	6:	IF bAWrappingCone23OnAuto AND bIWrappingChannelPiston2_End AND  bIWrappingChannelPiston3_End  AND NOT bAWrap_PistRsError
		AND bAFilmLoadedCom AND NOT bAConeMissErrorAtWrpConvTemp4_24  AND NOT bAConeMissErrorAtWrpConvTemp3_24  AND NOT
		 bAConeMissErrorAtWrpConvTemp2_24 AND NOT bAConeMissErrorAtWrpConvTemp5_24 AND b2_4SetHmiSelected
		AND NOT bQSealBitAlert (*AND NOT bQSealBitAlert_24*)   AND NOT SealConeMissAlet_24 THEN
		TON_8(IN:= FALSE);
		bAWrappingCone23FwdCom:=TRUE;
		bASensorMonitorBit2:=FALSE;
 		TON_6_24(IN:=FALSE) ;
		bWrapConvStopped3_24:=FALSE;
		TON_10_24(in:=FALSE);
		step3:=step3+1;
		ELSIF  bAWrappingCone23OnAuto AND bIWrappingChannelPiston2_End AND  bIWrappingChannelPiston3_End AND NOT bAWrap_PistRsError
		AND NOT bAFilmLoadedCom AND NOT bAPauseSeq THEN
		bAFlimNotLoaded2:=TRUE;
		bAWrappingCone23OnAuto:=FALSE;
		bAWrapConeCyl23_24_1:=FALSE;
		bAPolythinSheetError:=TRUE;
		bAConeMissErrorAtWrpConvTemp4_24:=FALSE;
		bWrapConvStopped3_24:=FALSE;
 		TON_6_24(IN:=FALSE);
		TON_10_24(in:=FALSE);
		bSheetNotFeeded:='Sheet NOT Feeded'; step3:=step3+3; END_IF

	7:	step3:=step3+1;

	8:	 IF bAWrappingCone23FwdCom AND NOT bAPauseSeq  THEN
		bAWrappingCone23OnAuto:=FALSE;
		bAFilmLoadedCom:=FALSE;
		bAConeMissErrorAtWrpConvTemp4_24:=FALSE;
		 TON_6_24(IN:=FALSE) ;
		bWrapConvStopped3_24:=FALSE;
		TON_10_24(in:=FALSE);
		step3:=step3+2;
		END_IF

	9:	 IF bFilmErrClear THEN bSheetNotFeeded:='Continue Machine Operation'; bAFlimNotLoaded2:=FALSE; bASensorMonitorBit2:=FALSE;  step3:=step3+1;END_IF

	10:	 IF NOT bAPauseSeq  THEN  bAWrapConeCyl23_24_1:=FALSE;
		bA6thConeWrappOver:=TRUE;
		step3:=step3+1; END_IF

	11:	bFilmErrClear:=FALSE; TON_6_24(IN:=FALSE) ;
		bWrapConvStopped3_24:=FALSE;
		TON_10_24(in:=FALSE);step3:=step3+1;

	12:	 IF bIWrappingChannelPiston2_Home AND    bIWrappingChannelPiston3_Home   THEN
		bASet3Comp:=TRUE;
		bASet2Comp:=FALSE;
		bAWrappingCone23FwdCom:=FALSE;
		b6thConePushed_24:=TRUE;
		bAFilm1Loaded_24_6Cone:=FALSE;
		bAFilm1Loaded_24_5Cone:=FALSE;
		bASensorMonitorBit2:=FALSE;
		bAConeMissErrorAtWrpConvTemp4_24:=FALSE;
		 TON_6_24(IN:=FALSE) ;
		TON_10_24(in:=FALSE);
		bWrapConvStopped3_24:=FALSE;
		bAWrapConeCyl23_24:=FALSE;
		step3:=0;
		END_IF    sMessage_Wrapping:='Check Wrapping Piston Home  2 & 3 Reed Switch';
END_CASE


IF bAFlimNotLoaded2 AND bErrorReset AND b2_4SetHmiSelected AND bAutoModeOn THEN step3:=10; bAFlimNotLoaded2:=FALSE;HmiFilmLoadErr:=''; END_IF




                                                                             (*===============Wrapping piston 23 (Cone7,8 )on/off logic  for 2*4 model====================*)


CASE step4 OF

	0:	TON_9(IN:= FALSE);
		step4:=step4+1;

	1:	 step4:=step4+1;

	2:	IF bAutoModeOn AND  bAWrapConeCyl23_24   AND SealingOver1  AND NOT bACheckWrappConvError5 AND NOT bAFlimNotLoaded2
		AND bIWrappingChannelPiston3_Home AND bIWrappingChannelPiston2_Home AND  b2_4SetHmiSelected AND NOT bAResetEnabled
		AND NOT bAConeMissErrorAtWrpConvTemp5_24   AND b2_4SetHmiSelected  AND SealingSafety THEN
		bA8thoneReachecdWCS:=TRUE;
		TON_9(IN:= TRUE, PT:=t#1s , Q=> , ET=> );
		 sMessage_Wrapping:='Check Wrapping Piston Home 2 & 3 Reed Switch';

		IF TON_9.Q THEN  SealingOver1:=FALSE; bASensorMonitorBit3:=FALSE; step4:=step4+1; END_IF
		END_IF

	3:	 step4:=step4+1;

	4:	IF NOT bQASealingConveyorMotor AND NOT bQSealBitAlert (*AND NOT bQSealBitAlert_24 *)AND  NOT bAPauseSeq  AND  bIWrappingCone2
		AND  bIWrappingCone3   AND NOT bAConeMissErrorAtWrpConvTemp5_24  AND b2_4SetHmiSelected  AND NOT SealConeMissAlet_24
		AND SealingSafety THEN
		bAWrappingCone23OnAuto1:=TRUE;
		step4:=step4+1;
		END_IF

	5:	 step4:=step4+1;

	6:	IF bAWrappingCone23OnAuto1 AND bIWrappingChannelPiston2_End AND  bIWrappingChannelPiston3_End  AND NOT bAWrap_PistRsError
		 AND bAFilmLoadedCom AND NOT bAConeMissErrorAtWrpConvTemp5_24  AND NOT bAConeMissErrorAtWrpConvTemp3_24
		 AND NOT bAConeMissErrorAtWrpConvTemp4_24  AND NOT bAConeMissErrorAtWrpConvTemp2_24 AND NOT bQSealBitAlert (*AND NOT bQSealBitAlert_24*)
		 AND NOT SealConeMissAlet_24 THEN
		TON_9(IN:= FALSE);
		bAWrappingCone23FwdCom1:=TRUE;
		bASensorMonitorBit3:=FALSE;
		TON_8_24(IN:=FALSE);
		TON_9_24(in:=FALSE);
		bWrapConvStopped4_24:=FALSE;
		step4:=step4+1;
		ELSIF bAWrappingCone23OnAuto1 AND bIWrappingChannelPiston2_End AND  bIWrappingChannelPiston3_End  AND NOT bAWrap_PistRsError
		 AND NOT  bAFilmLoadedCom AND NOT bAPauseSeq THEN
		bAFlimNotLoaded3:=TRUE;
		bAWrappingCone23OnAuto1:=FALSE;
		bAWrapConeCyl23_24:=FALSE;
		bAPolythinSheetError:=TRUE;
		bAConeMissErrorAtWrpConvTemp5_24:=FALSE;
		bWrapConvStopped4_24:=FALSE;
 		TON_8_24(IN:=FALSE);
		TON_9_24(in:=FALSE);
		bSheetNotFeeded:='Sheet NOT Feeded'; step4:=step4+3; END_IF


	7:	step4:=step4+1;

	8:	 IF bAWrappingCone23FwdCom1 AND NOT bAPauseSeq  THEN
		bAWrappingCone23OnAuto1:=FALSE;
		bAFilmLoadedCom:=FALSE;
		bAConeMissErrorAtWrpConvTemp5_24:=FALSE;
		TON_8_24(IN:=FALSE);
		TON_9_24(in:=FALSE);
		bWrapConvStopped4_24:=FALSE;
		step4:=step4+2;
		END_IF

	9:	 IF bFilmErrClear THEN bSheetNotFeeded:='Continue Machine Operation'; bAFlimNotLoaded3:=FALSE; bASensorMonitorBit3:=FALSE;  step4:=step4+1;END_IF

	10:	 IF NOT bAPauseSeq  THEN  bAWrapConeCyl23_24:=FALSE;
		bA8thConeWrappOver:=TRUE;
		step4:=step4+1; END_IF

	11:	bFilmErrClear:=FALSE; TON_8_24(IN:=FALSE);
		TON_9_24(in:=FALSE);
		bWrapConvStopped4_24:=FALSE;step4:=step4+1;


	12:	 IF    bIWrappingChannelPiston2_Home AND    bIWrappingChannelPiston3_Home   THEN
		bASet4Comp:=TRUE;
		bASet3Comp:=FALSE;
		bAWrappingCone23FwdCom1:=FALSE;
		b8thConesPushed:=TRUE;
		bAFilm1Loaded_24_8Cone:=FALSE;
		bAFilm1Loaded_24_7Cone:=FALSE;
		bASensorMonitorBit3:=FALSE;
		bAConeMissErrorAtWrpConvTemp5_24:=FALSE;
		TON_8_24(IN:=FALSE);
		bWrapConvStopped4_24:=FALSE;
		TON_9_24(in:=FALSE);
		bAWrapConeCyl23_24:=FALSE;
		step4:=0;
		END_IF   sMessage_Wrapping:='Check Wrapping Piston Home  2 & 3 Reed Switch';
END_CASE


IF bAFlimNotLoaded3 AND b2_4SetHmiSelected AND bErrorReset AND bAutoModeOn THEN step4:=10; bAFlimNotLoaded3:=FALSE;HmiFilmLoadErr:=''; END_IF






IF bA6conesPushed AND CounterTilt23.CV<=3 THEN
bANextLayerStarted:=TRUE;
END_IF


IF bA3Pushed OR bA6conesPushed AND bAFirstConeAtWrapConv THEN
bAConvStartInterlock:=TRUE;
ELSE
bAConvStartInterlock:=FALSE;
END_IF

(*

IF bAConvFirstStartUnitB THEN
baConveyerStarted:=TRUE;
END_IF
IF baConveyerStarted AND



*)




IF bIWrappingCone1 AND   InterLockCounter.CV = 0  AND NOT  bQWrappingConveyorMotor THEN
 Interlockfor_1Cone_24:=TRUE;
 ELSE
 Interlockfor_1Cone_24:=FALSE; END_IF


IF bIWrappingCone1 AND   InterLockCounter.CV = 4  AND NOT  bQWrappingConveyorMotor THEN
 Interlockfor_5Cone_24:=TRUE;
 ELSE
 Interlockfor_5Cone_24:=FALSE; END_IF

IF bIWrappingCone1 AND   InterLockCounter.CV = 6  AND NOT  bQWrappingConveyorMotor THEN
 Interlockfor_7Cone_24:=TRUE;
 ELSE
 Interlockfor_7Cone_24:=FALSE; END_IF

WrappingCone1RT(CLK:=( bIWrappingCone1 AND NOT Interlockfor_1Cone_24 AND NOT Interlockfor_5Cone_24 AND NOT Interlockfor_7Cone_24 ), Q=> );

WrappingConvRT(CLK:= bQWrappingConveyorMotor , Q=> );

IF  WrappingConvRT.Q THEN
bAWrapConvStarted:=TRUE;

END_IF

IF WrappingCone1RT.Q THEN WCS1Sensed:=TRUE; END_IF

IF WCS1Sensed  (* AND bAWrapConvStarted OR bConvRunning*)  THEN
bAInterlockCountStart:=TRUE;
ELSE
bAInterlockCountStart:=FALSE;
 END_IF


IF  bQWrappingConveyorMotor AND NOT bIWrappingCone1 AND bAutoModeOn THEN
WCS1Sensed:=FALSE;
END_IF

(*TON_6(IN:=WCS1Sensed , PT:=T#0.2s , Q=> , ET=> );

IF TON_6.Q THEN bAWrapConvStarted:=FALSE; (*TON_6(in:=FALSE);*)END_IF


IF InterLockCounter.CV = 2 AND bManualModeOn THEN
TimerStartBit:=TRUE;
bAWrapConvStarted:=FALSE;
TON_10(IN:=TimerStartBit , PT:=t#0.2s , Q=> , ET=> );

 END_IF


IF TON_10.Q AND bQWrappingConveyorMotor THEN
bConvRunning:=TRUE;(*TON_10(in:=FALSE);*)
END_IF*)




IF bRowStopperIntOver THEN
bSaelUnitIntOverTemp:=TRUE;
END_IF



                                                                   (*=============== Interlock Logic for  2*4 WCS conveyor===================*)


CASE step7 OF


	0:	IF bSaelUnitIntOverTemp AND b2_4SetHmiSelected  THEN                                    (*========= need to check for reset Logic=    step7:=0    =======*)
		Step7:=Step7+1;
		END_IF

	1:	bWCSStart1_24:=TRUE;
		Step7:=Step7+1;

	2:	IF  bASealConvEnd1_24 THEN
		bSaelUnitIntOverTemp:=FALSE;
		Step7:=Step7+1;
		END_IF

	3:	bWCSStart2_24:=TRUE;
		bASealConvEnd1_24:=FALSE;
		Step7:=Step7+1;


	4:	IF bASealConvEnd2_24  THEN
		Step7:=Step7+1;
		END_IF

	5:	bWCSStart3_24:=TRUE;
		bASealConvEnd2_24:=FALSE;
		Step7:=2;

END_CASE



IF NOT bIEmergencySwitch OR bStopHmi  OR bServoOff OR bIMcStop THEN

bAWrappingConvStartAuto3_23:=FALSE;
bAWrappingConvStartAuto4_23:=FALSE;
bAWrappingConvStartAuto3:=FALSE;
bAWrappingConvStartAuto4:=FALSE;
bAWrappingConvStartAuto5:=FALSE;


		bAWrappingCone123FwdCom:=FALSE;


SealingOver1:=FALSE;

bAFilm1Loaded:=FALSE;
bAFilm2Loaded:=FALSE;
bAFilm3Loaded:=FALSE;
		WrapConvStartDly(in:=FALSE);
		bAConvRunning1:=FALSE;
		bWrapConvStopped2:=FALSE;
		TON_3(IN:=FALSE);
		TON_13_24(in:=FALSE);
		TON_4_24(IN:=FALSE);
		TON_12_24(in:=FALSE);
		bAConeMissErrorAtWrpConvTemp1_24:=FALSE;
		bAConeMissErrorAtWrpConvTemp2_24:=FALSE;
		bAWrapConeCyl123:=FALSE;

bWrapConvStopped2:=FALSE;
bWrapConvStopped3_24:=FALSE;
bWrapConvStopped4_24:=FALSE;
bWrapConvStopped4_24exp:=FALSE;


bAWrappingConvStart1_23:=FALSE;
bAWrappingConvStart4_23:=FALSE;
bAWrappingConvStart1:=FALSE;
bAWrappingConvStart2:=FALSE;
bAWrappingConvStart3:=FALSE;
bAWrappingConvStart4:=FALSE;
bAWrappingConvStart5:=FALSE;

bAconvReayTemp:=FALSE;
bAconvReayTemp2:=FALSE;
bAconvReadyTemp3:=FALSE;
bAconvReadyTemp4:=FALSE;
bAconvReadyTemp5:=FALSE;

bAWrappingConvStart1_23:=FALSE;
bACheckWrappConvError1:=FALSE;
bACheckWrappConvError2:=FALSE;
bACheckWrappConvError3:=FALSE;
bACheckWrappConvError4:=FALSE;
bACheckWrappConvError5:=FALSE;

bAWrappingConvStartAuto:=FALSE;
bAWrappingConvStartAuto2:=FALSE;
 bAWrappingConvStartAuto3:=FALSE;

bQAWrappingConveyorMotor1:=FALSE;
 bQAWrappingConveyorMotor2:=FALSE;
bQAWrappingConveyorMotor3:=FALSE;
 bQAWrappingConveyorMotor4:=FALSE;
bQAWrappingConveyorMotor5:=FALSE;

WrapConvStartDly3_23(IN:= FALSE);

bAConvRunning1:=FALSE;
 bAConvStartBit:=FALSE;

bASensorMonitorBit1:=FALSE;
bASensorMonitorBit2:=FALSE;
 bASensorMonitorBit3:=FALSE;

bASet1Comp:=FALSE;
bASet3Comp:=FALSE;
bASet2Comp:=FALSE;
bASet4Comp:=FALSE;

bAWrapConeCyl3:=FALSE;
bAWrapConeCyl123:=FALSE;
bAWrapConeCyl23_24_1:=FALSE;
bAWrapConeCyl23_24:=FALSE;

WCS1Sensed:=FALSE;
bSaelUnitIntOver:=FALSE;


bASealConvEnd1:=FALSE;
bASealConvEnd2:=FALSE;

InterLockCounter.RESET:=TRUE;
bAWrappingCone123OnAuto:=FALSE;
bAWrappingCone123_23OnAuto:=FALSE;
bQAWrappingConveyorMotor4_23:=FALSE;
bQAWrappingConveyorMotor3_23:=FALSE;


bCount_ConvLockBit2:=FALSE;
bCount_ConvLockBit:=FALSE;
bASealConvEnd1_24:=FALSE;
bASealConvEnd2_24:=FALSE;
step1:=0;
step2:=0;
step3:=0;
step4:=0;
step5:=0;
step6:=0;
step7:=0;
bAConvStartBit:=FALSE;

bA3Pushed:=FALSE;
b4thConePushed:=FALSE;
b6thConePushed_24:=FALSE;

bWCSStart1_24:=FALSE;
bWCSStart2_24:=FALSE;
bWCSStart3_24:=FALSE;

TON_6_24(IN:=FALSE) ;

TON_8_24(IN:=FALSE) ;
TON_9_24(IN:=FALSE);
TON_10_24(IN:=FALSE);



		bAWrappingCone3FwdCom:=FALSE;
		bAFilm1Loaded_24_4Cone:=FALSE;
		bASensorMonitorBit1:=FALSE;
		bWrapConvStopped4_24exp:=FALSE;
 		TON_5_24(IN:=FALSE);
		TON_11_24(in:=FALSE);
		bAWrappingCone3OnAuto:=FALSE;
		bAFilmLoadedCom:=FALSE;
		bAConeMissErrorAtWrpConvTemp3_24:=FALSE;
		bWrapConvStopped4_24exp:=FALSE;
		bAWrapConeCyl3:=FALSE;
		bA4thWrappOver:=FALSE;

bAWrappingCone23FwdCom:=FALSE;
		bAFilm1Loaded_24_6Cone:=FALSE;
		bAFilm1Loaded_24_5Cone:=FALSE;
		bASensorMonitorBit2:=FALSE;
		bAConeMissErrorAtWrpConvTemp4_24:=FALSE;
		 TON_6_24(IN:=FALSE) ;
		TON_10_24(in:=FALSE);
		bWrapConvStopped3_24:=FALSE;
		bAWrapConeCyl23_24:=FALSE;
		bAWrapConeCyl23_24_1:=FALSE;
		bA6thConeWrappOver:=FALSE;


		bAWrappingCone23FwdCom1:=FALSE;
		b8thConesPushed:=FALSE;
		bAFilm1Loaded_24_8Cone:=FALSE;
		bAFilm1Loaded_24_7Cone:=FALSE;
		bASensorMonitorBit3:=FALSE;
		bAConeMissErrorAtWrpConvTemp5_24:=FALSE;
		TON_8_24(IN:=FALSE);
		bWrapConvStopped4_24:=FALSE;
		TON_9_24(in:=FALSE);
		bAWrapConeCyl23_24:=FALSE;
		bAWrapConeCyl23_24:=FALSE;
		bA8thConeWrappOver:=FALSE;

ELSE
InterLockCounter.RESET:=FALSE;
END_IF
END_PROGRAM

(* POU Auto/Sealing_Conveyor_24, ST *)
PROGRAM Sealing_Conveyor_24
VAR
	bA3ConeSealStarted: BOOL;
	bA3ConeSealComp: BOOL;

	bAConeCountSenEnable1: BOOL;
	CTU_1: CTU;
	step1: INT;
	step2: INT;
	bA4thConeSealStarted: BOOL;
	bA4thConeSealComp: BOOL;

	ConvStopDly1: TON;
	bAColoumnConeDeducted: BOOL;
	step3: INT;
	bA6thConeSealStarted: BOOL;
	bA6thConeSealComp: BOOL;

	ConvStopDly2: TON;
	ConvStopDly3: TON;
	bA8thConeSealStarted: BOOL;
	bA8thConeSealComp: BOOL;
	step4: INT;

	ConvStopDly4: TON;
	bQASealingConveyor1: BOOL;
	bQASealingConveyor2: BOOL;
	bQASealingConveyor3: BOOL;
	bQASealingConveyor4: BOOL;
	Step5: INT;
	bSealConvIntOverTemp: BOOL;
	CTU_1AlarmOnly: CTU;

	bCountLockBit_24: BOOL;
	CTU_1_24: CTU;
	CTU_1_24_AlarmOnly: CTU;
	bQASealingConveyor5: BOOL;
	bQASealingConveyor6: BOOL;
	bQASealingConveyor7: BOOL;
	bQASealingConveyor8: BOOL;
	bSecSetStarted_24: BOOL;
	SealCountBit_24: BOOL;
	bCountLock1: BOOL;
	bCountLock5_24: BOOL;
	bCountLock6_24: BOOL;
	bCountLock2_24: BOOL;
	bCountLock3_24: BOOL;
	bCountLock4_24: BOOL;
	bCountLock1_24: BOOL;
	bCountLock7_24: BOOL;
	bCountLock8_24: BOOL;
	bCountLock: BOOL;
	bAConeMissAtSealConv4_24: BOOL;
	tSealStopDly_24: TIME;
	bAConeMissAtSealConv1_24: BOOL;
	bAConeMissAtSealConv2_24: BOOL;
	bAConeMissAtSealConv3_24: BOOL;
	bQASealingConveyor9: BOOL;
	bAConeMissAtSealConv5_24: BOOL;
	Timer1: TON;
	bA4ConeCrossed_24: BOOL;
	bA6ConeCrossed_24: BOOL;
	bA8ConeCrossed_24: BOOL;
	ConvStopDly01_24: TON;
	bQASealingConveyor123_24: BOOL;
	bQASealingConveyor1234_24: BOOL;
	ConvStopDly02_24: TON;
	ConvStopDly03_24: TON;
	ConvStopDly04_24: TON;
	bQASealingConveyor123456_24: BOOL;
	bQASealingConveyor12345678_24: BOOL;
	bQASealingConveyor10: BOOL;
	bQASealingConveyor11: BOOL;
	bAConeMissAtSealConv6_24: BOOL;
	bAConeMissAtSealConv7_24: BOOL;
	bQASealingConveyor12: BOOL;
	bAConeMissAtSealConv8_24: BOOL;
	bCountLock10_24: BOOL;
	bCountLock9_24: BOOL;
	bCountLock123_24: BOOL;
	bCountLock1234_24: BOOL;
	ConvStopDly06_24: TON;
	bQASealingConveyor1234_24_1: BOOL;
	bQASealingConveyor123_24_1: BOOL;
	ConvStopDly07_24: TON;
	ConvStopDly08_24: TON;
	bQASealingConveyor123456_24_1: BOOL;
	ConvStopDly09_24: TON;
	bQASealingConveyor12345678_24_1: BOOL;
	ConvStopDly11_24: TON;
	bQASealingConveyorSample123_24: BOOL;
	bQASealingConveyorSample1234_24: BOOL;
	bQASealingConveyorSample123456_24: BOOL;
	bQASealingConveyorSample12345678_24: BOOL;
	bCountLock_24: BOOL;
	bCountLock123_24_1: BOOL;
	bCountLock1234_24_1: BOOL;
	bCountLock123456_24_1: BOOL;
	bCountLock11_24: BOOL;
	bCountLock123456_24: BOOL;
	bCountLock12345678_24_1: BOOL;
	bCountLock12_24: BOOL;
	bCountLock12345678_24: BOOL;
	bSet1Started_24: BOOL;
	bSet2Started_24: BOOL;
	bSet3Started_24: BOOL;
	bSet4Started_24: BOOL;
	bCountLockBit1_24: BOOL;
	bCountLockBit2_24: BOOL;
	bCountLockBit3_24: BOOL;
	bCountLockBit4_24: BOOL;
	bAConeMissAtSealConv01_24: BOOL;
	bACounter_24Reset: BOOL;
	bACounter_24: BOOL;
END_VAR
							(*###########################Sealing Conveyor On Bit######################### *)

bQASealingConveyorMotor1:= (bQASealingConveyor1 OR bQASealingConveyor2 OR bQASealingConveyor3 OR bQASealingConveyor4 OR bQASealingConveyor5 OR bQASealingConveyor6 OR bQASealingConveyor7 OR bQASealingConveyor8 OR bQASealingConveyor9 OR bQASealingConveyor10 OR bQASealingConveyor11 OR bQASealingConveyor12 );

							(*###########################Sealing Conveyor Count interlock t######################### *)

IF bQASealingConveyorMotor AND bSet1Started_24  AND CTU_1_24_AlarmOnly.CV=3 THEN bCountLockBit1_24:=TRUE; END_IF
IF bQASealingConveyorMotor AND bSet2Started_24  AND CTU_1_24_AlarmOnly.CV=4 THEN bCountLockBit2_24:=TRUE; END_IF
IF bQASealingConveyorMotor AND bSet3Started_24  AND CTU_1_24_AlarmOnly.CV=6 THEN bCountLockBit3_24:=TRUE; END_IF
IF bQASealingConveyorMotor AND bSet4Started_24  AND CTU_1_24_AlarmOnly.CV=8 THEN bCountLockBit4_24:=TRUE; END_IF


IF bQASealingConveyorMotor AND bIConeCountSensor AND b2_4SetHmiSelected  AND NOT bCountLockBit1_24 AND NOT bCountLockBit2_24
 AND NOT bCountLockBit3_24 AND NOT bCountLockBit4_24  THEN
	bAConeCountSenEnable1:=TRUE;
ELSE
	bAConeCountSenEnable1:=FALSE;
END_IF

CTU_1(
	CU:=bAConeCountSenEnable1 ,
	RESET:= ,
	PV:=8 ,
	Q=> ,
	CV=> );


CTU_1_24_AlarmOnly(
	CU:=(bAConeCountSenEnable1 AND NOT bCountLock_24) ,
	RESET:=bACounter_24Reset OR bACounter_24 ,
	PV:=8 ,
	Q=> ,
	CV=> );


IF bQASealingConveyorMotor AND bSecSetStarted_24 AND  CTU_1.CV=8 THEN SealCountBit_24:=TRUE; END_IF


				(*############################  1,2,3rd  Cone Sealing Conveyor   ############################*)


CASE step1 OF

		0:	IF bAutoModeOn AND b2_4SetHmiSelected AND  bA3ConeWrappOver_24 AND bQASealingSeparatorYAxisPistonValve THEN
			bA3ConeSealStarted:=TRUE;
			CTU_1.RESET:=TRUE;
			bACounter_24:=TRUE;
			 tSealStopDly_24:=t#2.5s;
			ConvStopDly1(IN:=FALSE); ConvStopDly06_24(in:=FALSE);
			 step1:=step1+1; END_IF

		1:	IF NOT bAPauseSeq THEN step1:=step1+1; END_IF

		2:	IF bAutoModeOn AND b2_4SetHmiSelected AND  bA3ConeSealStarted AND bISealingSeparatorXAxisEnd THEN
			bA3ConeSealComp:=TRUE;
			CTU_1.RESET:=FALSE;
			bACounter_24:=FALSE;
		 	Timer1(IN:=FALSE);
			step1:=step1+1; END_IF

		3:	IF NOT bAPauseSeq THEN step1:=step1+1; END_IF

		4:	IF bAutoModeOn AND   bA3ConeSealComp AND (bSealConvStart1_24 OR bSealConvStart3_24)  AND NOT bASealSepaX_axisRsError THEN
			bQASealingConveyor1:=TRUE;
			ConvStopDly1(in:=FALSE);
			ConvStopDly06_24(in:=FALSE);
			bSet1Started_24:=TRUE;
			 step1:=step1+1; END_IF

		5:	ConvStopDly1(in:=FALSE);
			 step1:=step1+1;

		6:	IF NOT bAPauseSeq THEN  step1:=step1+1; END_IF

		7:	IF CTU_1_24_AlarmOnly.CV>=3 THEN
			bSealConvStart1_24:=FALSE;
			bSealConvStart3_24:=FALSE;
			bA3ConeCrossed_24:=TRUE;
			bA3ConeSealComp:=FALSE;
			bA3ConeSealStarted:=FALSE;
			 step1:=step1+1; END_IF

		8:	IF bIColumnconeDetection THEN
		step1:=step1+1;
		END_IF

		9:	ConvStopDly1(IN:=TRUE , PT:= t#0.5s , Q=> , ET=> );
			IF ConvStopDly1.Q THEN step1:=step1+1; END_IF

		10:	 step1:=step1+1;

		11:	bQASealingConveyor1:=FALSE;
			bQASealingConveyor5:=FALSE;
			bQASealingConveyor6:=FALSE;
			bA3ConeSealComp:=FALSE;
			bA3ConeSealStarted:=FALSE;
			bCountLock1_24:=FALSE;
			bCountLock5_24:=FALSE;
			bCountLock6_24:=FALSE;
			bA3ConeCrossed_24:=FALSE;
			bQASealingConveyor123_24:=FALSE;
			bAConeMissAtSealConv2_24:=FALSE;
			ConvStopDly01_24(in:=FALSE);
			bQASealingConveyorSample123_24:=FALSE;
			bQASealingConveyor123_24_1:=FALSE;
			bSet1Started_24:=FALSE;
			bCountLockBit1_24:=FALSE;
			bCountLock123_24:=FALSE;
			bCountLock123_24_1:=FALSE;
			ConvStopDly06_24(in:=FALSE);
			step1:=step1+1;


		12:	IF NOT bAPauseSeq THEN step1:=step1+1; END_IF

		13:	step1:=0;

END_CASE

				(*############################  4th Cone Sealing Conveyor   #####################*)

CASE step2 OF

	0:	IF bAutoModeOn AND b2_4SetHmiSelected AND  bA4thWrappOver AND bQASealingSeparatorYAxisPistonValve THEN
		bA4thConeSealStarted:=TRUE;
		 tSealStopDly_24:=t#2.5s;
		ConvStopDly2(IN:=FALSE);
		bQASealingConveyor123_24_1:=FALSE;
		ConvStopDly06_24(in:=FALSE);
		step2:=step2+1;
		END_IF

	1:	IF NOT bAPauseSeq THEN step2:=step2+1; END_IF

	2:	IF bAutoModeOn AND b2_4SetHmiSelected AND  bA4thConeSealStarted AND bISealingSeparatorXAxisEnd THEN
		bA4thConeSealComp:=TRUE;
		step2:=step2+1;
		END_IF

	3:	IF NOT bAPauseSeq THEN step2:=step2+1; END_IF

	4:	IF bAutoModeOn AND   bA4thConeSealComp  AND NOT bAPauseSeq THEN
		bQASealingConveyor2:=TRUE;
		bSet2Started_24:=TRUE;
		step2:=step2+1;
		END_IF

	5:	ConvStopDly2(in:=FALSE);
		ConvStopDly07_24(in:=FALSE);
		step2:=step2+1;

	6:	IF NOT bAPauseSeq THEN step2:=step2+1; END_IF

	7:	IF CTU_1_24_AlarmOnly.CV>=4 THEN
		bA4thConeSealComp:=FALSE;
		bA4thConeSealStarted:=FALSE;
		bA4ConeCrossed_24:=TRUE;
		step2:=step2+1;
		END_IF

	8:	IF NOT bAPauseSeq THEN step2:=step2+1; END_IF

	9:	IF bIColumnconeDetection THEN
		ConvStopDly2(IN:=TRUE , PT:=t#2s , Q=> , ET=> );
		IF ConvStopDly2.Q THEN    step2:=step2+1; END_IF
		END_IF

	10:	 step2:=step2+1;

	11:	bQASealingConveyor2:=FALSE;
		bQASealingConveyor9:=FALSE;
		bAColumnPushPistonStart1:=TRUE;
		bASealConvEnd1_24:=TRUE;
		bA4ConeCrossed_24:=FALSE;
		bQASealingConveyor1234_24:=FALSE;
		bAConeMissAtSealConv3_24:=FALSE;
		bAConeMissAtSealConv4_24:=FALSE;
		bQASealingConveyor10:=FALSE;
		ConvStopDly02_24(in:=FALSE);
		bQASealingConveyor9:=FALSE;
		ConvStopDly07_24(in:=FALSE);
		bQASealingConveyorSample1234_24:=FALSE;
		bQASealingConveyor1234_24_1:=FALSE;
		bSet2Started_24:=FALSE;
		bCountLockBit2_24:=FALSE;
		bCountLock1234_24_1:=FALSE;
		bCountLock1234_24:=FALSE;
		bCountLock2_24:=FALSE;
		bCountLock9_24:=FALSE;
		bCountLock10_24:=FALSE;
		step2:=0;


END_CASE


				(*############################  5,6th Cone Sealing Conveyor   #########################*)


CASE step3 OF

	0:	IF bAutoModeOn AND b2_4SetHmiSelected AND  bA6thConeWrappOver AND bQASealingSeparatorYAxisPistonValve THEN
		bA6thConeSealStarted:=TRUE;
		 tSealStopDly_24:=t#2.5s;
		ConvStopDly3(IN:=FALSE );
		bQASealingConveyor1234_24_1:=FALSE;
		ConvStopDly07_24(in:=FALSE);
		step3:=step3+1;
		END_IF

	1:	IF NOT bAPauseSeq THEN step3:=step3+1; END_IF

	2:	IF bAutoModeOn AND b2_4SetHmiSelected AND  bA6thConeSealStarted AND bISealingSeparatorXAxisEnd THEN
		bA6thConeSealComp:=TRUE;
		step3:=step3+1;
		END_IF

	3:	IF NOT bAPauseSeq THEN step3:=step3+1; END_IF

	4:	IF bAutoModeOn AND   bA6thConeSealComp AND bSealConvStart2_24 AND NOT bAPauseSeq  THEN
		bQASealingConveyor3:=TRUE;
		bSet3Started_24:=TRUE;
		step3:=step3+1;
		END_IF


	5:	ConvStopDly3(in:=FALSE);
		ConvStopDly08_24(in:=FALSE);
 		step3:=step3+1;


	6:	IF NOT bAPauseSeq THEN step3:=step3+1; END_IF

	7:	IF CTU_1_24_AlarmOnly.CV>=6 THEN
		bSealConvStart2_24:=FALSE;
		bA6ConeCrossed_24:=TRUE;
		ConvStopDly3(IN:=TRUE , PT:=t#0.5s , Q=> , ET=> );
		IF ConvStopDly3.Q THEN  step3:=step3+1; END_IF
		END_IF

	8:	 step3:=step3+1;

	9:	bA6thConeSealComp:=FALSE;
		bA6thConeSealStarted:=FALSE;
		bQASealingConveyor3:=FALSE;
		bQASealingConveyor7:=FALSE;
		bA6ConeCrossed_24:=FALSE;
		bQASealingConveyor123456_24:=FALSE;
		bAConeMissAtSealConv4_24:=FALSE;
		ConvStopDly03_24(in:=FALSE);
		bAConeMissAtSealConv6_24:=FALSE;
		bQASealingConveyor11:=FALSE;
		ConvStopDly08_24(in:=FALSE);
		bQASealingConveyorSample123456_24:=FALSE;
		bSet3Started_24:=FALSE;
		bCountLockBit3_24:=FALSE;
		bCountLock3_24:=FALSE;
		bCountLock7_24:=FALSE;
		bCountLock11_24:=FALSE;
		bCountLock123456_24:=FALSE;
		bCountLock123456_24_1:=FALSE;
		bQASealingConveyor123456_24_1:=FALSE;
		step3:=step3+1;

	10:	IF NOT bAPauseSeq THEN step3:=step3+1; END_IF

	11:	step3:=0;

END_CASE


				(*############################  7, 8th Cone Sealing Conveyor   #########################*)


CASE step4 OF

	0:	IF bAutoModeOn AND b2_4SetHmiSelected AND  bA8thConeWrappOver AND bQASealingSeparatorYAxisPistonValve THEN
		bA8thConeSealStarted:=TRUE;
		 tSealStopDly_24:=t#2.5s;
		ConvStopDly4(IN:=FALSE);
		step4:=step4+1;
		END_IF

	1:	IF NOT bAPauseSeq THEN step4:=step4+1; END_IF

	2:	IF bAutoModeOn AND b2_4SetHmiSelected AND  bA8thConeSealStarted AND bISealingSeparatorXAxisEnd THEN
		bA8thConeSealComp:=TRUE;
		step4:=step4+1;
		END_IF

	3:	IF NOT bAPauseSeq THEN step4:=step4+1; END_IF

	4:	IF bAutoModeOn AND   bA8thConeSealComp AND NOT bAPauseSeq   THEN
		bQASealingConveyor4:=TRUE;
		bSet4Started_24:=TRUE;
		step4:=step4+1;
		END_IF

	5:	ConvStopDly4(in:=FALSE);
		ConvStopDly11_24(in:=FALSE);
 		step4:=step4+1;

	6:	IF NOT bAPauseSeq THEN step4:=step4+1; END_IF

	7:	IF CTU_1_24_AlarmOnly.CV=8 THEN
		bA8thConeSealComp:=FALSE;
		bA8thConeSealStarted:=FALSE;
		bA8ConeCrossed_24:=TRUE;
		step4:=step4+1;
		END_IF

	8:	IF NOT bAPauseSeq THEN step4:=step4+1; END_IF

	9:	IF bIColumnconeDetection THEN
		ConvStopDly4(IN:=TRUE , PT:=tSealStopDly_24 , Q=> , ET=> );
		IF ConvStopDly4.Q THEN  bACounter_24:=TRUE;   step4:=step4+1; END_IF
		END_IF

	10:	 step4:=step4+1;

	11:	bQASealingConveyor4:=FALSE;
		bQASealingConveyor8:=FALSE;
		bAColumnPushPistonStart2:=TRUE;
		bASealConvEnd2_24:=TRUE;
		CTU_1.RESET:=FALSE;
		SealCountBit_24:=FALSE;
		bA8ConeCrossed_24:=FALSE;
		bQASealingConveyor12345678_24:=FALSE;
		ConvStopDly04_24(in:=FALSE);
		bAConeMissAtSealConv7_24:=FALSE;
		bQASealingConveyor12:=FALSE;
		bAConeMissAtSealConv8_24:=FALSE;
		ConvStopDly11_24(in:=FALSE);
		bQASealingConveyor12345678_24_1:=FALSE;
		bQASealingConveyorSample12345678_24:=FALSE;
		bSet4Started_24:=FALSE;
		bCountLockBit4_24:=FALSE;
		bCountLock4_24:=FALSE;
		bCountLock8_24:=FALSE;
		bCountLock12_24:=FALSE;
		bCountLock12345678_24:=FALSE;
		bCountLock12345678_24_1:=FALSE;
		step4:=0;
		bACounter_24:=FALSE;
END_CASE




IF bRowStopperIntOver  AND b2_4SetHmiSelected THEN
bSealConvIntOverTemp:=TRUE;
END_IF


CASE step5 OF


0:	IF bSealConvIntOverTemp  AND b2_4SetHmiSelected THEN
	Step5:=Step5+1;
	END_IF

1:	IF NOT bIColumnconeDetection THEN
	bSealConvStart1_24:=TRUE;
	Step5:=Step5+1;
	END_IF

2:	IF  CTU_1_24_AlarmOnly.CV=4 THEN

	Step5:=Step5+1;
	END_IF

3:	IF bIColumnconeDetection THEN
	Step5:=Step5+1;
	END_IF

4:	IF bAFirstSetToMatrix  THEN
	bSealConvStart2_24:=TRUE;
	Step5:=Step5+1;
	END_IF

5:	IF	CTU_1_24_AlarmOnly.CV=8 THEN
	bAFirstSetToMatrix:=FALSE;
	Step5:=Step5+1;
	END_IF

6:	IF bIColumnconeDetection THEN
	Step5:=Step5+1;
	END_IF

7:	IF bASecondSetToMatrix THEN
	bSealConvStart3_24:=TRUE;
	Step5:=Step5+1;
	END_IF

8:	bASecondSetToMatrix:=FALSE;
	Step5:=1;
END_CASE


(*

	IF bAresetHmi THEN
	Step5:=0;
	bSealConvStart1_24:=FALSE;
	bSealConvStart2_24:=FALSE;
	bASecondSetToMatrix:=FALSE;
	bAFirstSetToMatrix:=FALSE;
	bSealConvStart3_24:=FALSE;
	END_IF
*)

									(*--------------------------------------------------------Alarm Sequence---------------------------------------------------------*)

IF bQASealingConveyor1 AND CTU_1_24_AlarmOnly.CV =3  THEN  bCountLock1_24:=TRUE; END_IF
IF bQASealingConveyor5 AND CTU_1_24_AlarmOnly.CV =3  THEN  bCountLock5_24:=TRUE; END_IF
IF bQASealingConveyor6 AND CTU_1_24_AlarmOnly.CV =3  THEN  bCountLock6_24:=TRUE; END_IF
IF bQASealingConveyor123_24	   AND CTU_1_24_AlarmOnly.CV=3 THEN  bCountLock123_24:=TRUE; END_IF
IF bQASealingConveyor123_24_1 AND CTU_1_24_AlarmOnly.CV=3 THEN bCountLock123_24_1:=TRUE;END_IF


IF bQASealingConveyor2 AND CTU_1_24_AlarmOnly.CV =4  THEN  bCountLock2_24:=TRUE; END_IF
IF bQASealingConveyor10 AND CTU_1_24_AlarmOnly.CV =4  THEN  bCountLock10_24:=TRUE; END_IF
IF bQASealingConveyor1234_24_1 AND CTU_1_24_AlarmOnly.CV =4 THEN bCountLock1234_24_1:=TRUE; END_IF
IF bQASealingConveyor9 AND CTU_1_24_AlarmOnly.CV =4  THEN  bCountLock9_24:=TRUE; END_IF
IF bQASealingConveyor1234_24 AND CTU_1_24_AlarmOnly.CV =4  THEN  bCountLock1234_24:=TRUE; END_IF


IF bQASealingConveyor3 AND CTU_1_24_AlarmOnly.CV =6  THEN  bCountLock3_24:=TRUE; END_IF
IF bQASealingConveyor7 AND CTU_1_24_AlarmOnly.CV =6  THEN  bCountLock7_24:=TRUE; END_IF
IF bQASealingConveyor123456_24_1 AND CTU_1_24_AlarmOnly.CV =6  THEN  bCountLock123456_24_1:=TRUE; END_IF
IF bQASealingConveyor11 AND CTU_1_24_AlarmOnly.CV =6  THEN  bCountLock11_24:=TRUE; END_IF
IF bQASealingConveyor123456_24 AND CTU_1_24_AlarmOnly.CV =6  THEN  bCountLock123456_24:=TRUE; END_IF

IF bQASealingConveyor4 AND CTU_1_24_AlarmOnly.CV =8  THEN  bCountLock4_24:=TRUE; END_IF
IF bQASealingConveyor12345678_24_1 AND CTU_1_24_AlarmOnly.CV =8  THEN  bCountLock12345678_24_1:=TRUE; END_IF
IF bQASealingConveyor12 AND CTU_1_24_AlarmOnly.CV =8  THEN  bCountLock12_24:=TRUE; END_IF
IF bQASealingConveyor12345678_24 AND CTU_1_24_AlarmOnly.CV =8  THEN  bCountLock12345678_24:=TRUE; END_IF
IF bQASealingConveyor8 AND CTU_1_24_AlarmOnly.CV =8  THEN  bCountLock8_24:=TRUE; END_IF

 IF bCountLock1_24 OR bCountLock2_24 OR  bCountLock3_24 OR bCountLock4_24 OR  bCountLock5_24 OR bCountLock6_24
OR bCountLock7_24 OR bCountLock8_24 OR bCountLock9_24 OR bCountLock10_24 OR bCountLock11_24 OR bCountLock12_24
OR bCountLock123_24 OR  bCountLock1234_24  OR  bCountLock123456_24 OR  bCountLock12345678_24
OR bCountLock123_24_1 OR bCountLock1234_24_1 OR bCountLock123456_24_1 OR bCountLock12345678_24_1
THEN
 bCountLock_24:=TRUE;
 ELSE
bCountLock_24:=FALSE;
 END_IF

						(*--------------------------------------------------------Alarm Sequence Cone 2 Missing---------------------------------------------------------*)


IF bQASealingConveyor1 AND NOT bIConeCountSensor AND  NOT bAPauseSeq  THEN ConvStopDly06_24(IN:=TRUE , PT:=t#6s , Q=> , ET=> );END_IF
IF ConvStopDly06_24.Q THEN bQASealingConveyor123_24_1:=TRUE; bQASealingConveyor1:=FALSE; END_IF

IF bQASealingConveyor123_24_1    AND  (CTU_1_24_AlarmOnly.CV ) <3  AND  NOT bAPauseSeq THEN
bAConeMissAtSealConv01_24:=TRUE;
bQASealingConveyor1:=FALSE;
bQASealingConveyor123_24_1:=FALSE;
ConvStopDly06_24(in:=FALSE);
SealConeMiss:=' Cone  Missing From Sealing Conveyor';
END_IF
IF bAConeMissAtSealConv01_24 AND bErrorReset THEN
bQASealingConveyor5:=TRUE;
bAConeMissAtSealConv01_24:=FALSE;
Step1:=5;  (*tSealStopDly_24:=t#4s;*)
SealConeMiss:='Continue Machine Operation'; END_IF



						(*--------------------------------------------------------Alarm Sequence Cone 3 Missing---------------------------------------------------------*)



IF bQASealingConveyor5 OR bQASealingConveyor123_24    AND  (CTU_1_24_AlarmOnly.CV ) <3  AND  NOT bAPauseSeq  THEN
bAConeMissAtSealConv2_24:=TRUE;
bQASealingConveyor5:=FALSE;
bQASealingConveyor6:=FALSE;
bQASealingConveyor123_24:=FALSE;
ConvStopDly01_24(in:=FALSE);
bQASealingConveyorSample123_24:=FALSE;
SealConeMiss:=' Cone  Missing From Sealing Conveyor';
 END_IF
IF bAConeMissAtSealConv2_24 AND bErrorReset THEN
bQASealingConveyor6:=TRUE;  Step1:=5;  tSealStopDly_24:=t#4s;
SealConeMiss:='Continue Machine Operation'; bAConeMissAtSealConv2_24:=FALSE; END_IF

IF bQASealingConveyor6 THEN ConvStopDly01_24(IN:=TRUE , PT:=t#6s , Q=> , ET=> ); bQASealingConveyorSample123_24:=TRUE; END_IF
IF ConvStopDly01_24.Q THEN bQASealingConveyor123_24:=TRUE; END_IF



					(*--------------------------------------------------------Alarm Sequence Cone 4 Missing---------------------------------------------------------*)



IF bQASealingConveyor2 AND NOT bIConeCountSensor  AND  NOT bAPauseSeq THEN ConvStopDly07_24(IN:=TRUE , PT:=t#5s , Q=> , ET=> ); END_IF
IF ConvStopDly07_24.Q THEN bQASealingConveyor1234_24_1:=TRUE; bQASealingConveyor2:=FALSE; END_IF

IF bQASealingConveyor1234_24_1  AND  bIColumnconeDetection  AND  (CTU_1_24_AlarmOnly.CV ) <4  AND(CTU_1_24_AlarmOnly.CV ) =3 AND  NOT bAPauseSeq THEN
bAConeMissAtSealConv3_24:=TRUE;
bQASealingConveyor2:=FALSE;
bQASealingConveyor1234_24_1:=FALSE;
ConvStopDly07_24(in:=FALSE);
SealConeMiss:=' Cone  Missing From Sealing Conveyor';
END_IF
IF bAConeMissAtSealConv3_24 AND bErrorReset THEN
bQASealingConveyor10:=TRUE;
bAConeMissAtSealConv3_24:=FALSE;
Step2:=5;  tSealStopDly_24:=t#4s;
SealConeMiss:='Continue Machine Operation'; END_IF


IF bQASealingConveyor10 OR bQASealingConveyor1234_24 AND  bIColumnconeDetection  AND  (CTU_1_24_AlarmOnly.CV ) <4 AND (CTU_1_24_AlarmOnly.CV ) =3 AND  NOT bAPauseSeq   THEN
bAConeMissAtSealConv4_24:=TRUE;
bQASealingConveyor10:=FALSE;
bQASealingConveyor1234_24:=FALSE;
ConvStopDly02_24(in:=FALSE);
bQASealingConveyor9:=FALSE;
bQASealingConveyorSample1234_24:=FALSE;
SealConeMiss:=' Cone  Missing From Sealing Conveyor';
 END_IF
IF bAConeMissAtSealConv4_24 AND bErrorReset THEN
bQASealingConveyor9:=TRUE;  Step2:=5;  tSealStopDly_24:=t#4s;
SealConeMiss:='Continue Machine Operation'; bAConeMissAtSealConv4_24:=FALSE; END_IF

IF bQASealingConveyor9 THEN ConvStopDly02_24(IN:=TRUE , PT:=t#6s , Q=> , ET=> ); bQASealingConveyorSample1234_24:=TRUE;END_IF
IF ConvStopDly02_24.Q THEN bQASealingConveyor1234_24:=TRUE; END_IF



					(*--------------------------------------------------------Alarm Sequence Cone 6 Missing---------------------------------------------------------*)


IF bQASealingConveyor3 AND NOT bIConeCountSensor  AND  NOT bAPauseSeq THEN ConvStopDly08_24(IN:=TRUE , PT:=t#5s , Q=> , ET=> ); END_IF
IF ConvStopDly08_24.Q THEN bQASealingConveyor123456_24_1:=TRUE; bQASealingConveyor3:=FALSE; END_IF

IF bQASealingConveyor123456_24_1    AND  (CTU_1_24_AlarmOnly.CV ) <6  AND  (CTU_1_24_AlarmOnly.CV ) >=4  AND  NOT bAPauseSeq THEN
bAConeMissAtSealConv5_24:=TRUE;
bQASealingConveyor3:=FALSE;
ConvStopDly08_24(in:=FALSE);
bQASealingConveyor123456_24_1:=FALSE;
SealConeMiss:=' Cone  Missing From Sealing Conveyor';
END_IF
IF bAConeMissAtSealConv5_24 AND bErrorReset THEN
bQASealingConveyor11:=TRUE;
bAConeMissAtSealConv5_24:=FALSE;
Step3:=5;  tSealStopDly_24:=t#4s;
SealConeMiss:='Continue Machine Operation';
END_IF

IF bQASealingConveyor11  OR bQASealingConveyor123456_24   AND  (CTU_1_24_AlarmOnly.CV ) <6 AND  (CTU_1_24_AlarmOnly.CV ) >=4 AND  NOT bAPauseSeq   THEN
bAConeMissAtSealConv6_24:=TRUE;
bQASealingConveyor11:=FALSE;
bQASealingConveyor123456_24:=FALSE;
ConvStopDly03_24(in:=FALSE);
bQASealingConveyor7:=FALSE;
bQASealingConveyorSample123456_24:=FALSE;
SealConeMiss:=' Cone  Missing From Sealing Conveyor';
 END_IF
IF bAConeMissAtSealConv6_24 AND bErrorReset THEN
bQASealingConveyor7:=TRUE;  Step3:=5;  tSealStopDly_24:=t#4s;
SealConeMiss:='Continue Machine Operation'; bAConeMissAtSealConv6_24:=FALSE; END_IF

IF bQASealingConveyor7 THEN ConvStopDly03_24(IN:=TRUE , PT:=t#6s , Q=> , ET=> ); bQASealingConveyorSample123456_24:=TRUE;END_IF
IF ConvStopDly03_24.Q THEN bQASealingConveyor123456_24:=TRUE; END_IF


		                            (*--------------------------------------------------------Alarm Sequence Cone 8 Missing---------------------------------------------------------*)


IF bQASealingConveyor4 AND NOT bIConeCountSensor  AND  NOT bAPauseSeq THEN ConvStopDly11_24(IN:=TRUE , PT:=t#5s , Q=> , ET=> ); END_IF
IF ConvStopDly11_24.Q THEN bQASealingConveyor12345678_24_1:=TRUE; bQASealingConveyor4:=FALSE; END_IF


IF bQASealingConveyor12345678_24_1  AND  bIColumnconeDetection  AND  (CTU_1_24_AlarmOnly.CV ) <8 AND  (CTU_1_24_AlarmOnly.CV ) >=6  AND  NOT bAPauseSeq THEN
bAConeMissAtSealConv7_24:=TRUE;
bQASealingConveyor4:=FALSE;
ConvStopDly11_24(in:=FALSE);
bQASealingConveyor12345678_24_1:=FALSE;
SealConeMiss:=' Cone  Missing From Sealing Conveyor';
END_IF
IF bAConeMissAtSealConv7_24 AND bErrorReset THEN
bQASealingConveyor12:=TRUE;
bAConeMissAtSealConv7_24:=FALSE;
Step4:=5;  tSealStopDly_24:=t#4s;
SealConeMiss:='Continue Machine Operation'; END_IF


IF bQASealingConveyor12 OR bQASealingConveyor12345678_24  AND  bIColumnconeDetection  AND  (CTU_1_24_AlarmOnly.CV ) <8 AND  (CTU_1_24_AlarmOnly.CV ) >=6
AND  NOT bAPauseSeq THEN
bAConeMissAtSealConv8_24:=TRUE;
bQASealingConveyor12:=FALSE;
bQASealingConveyor12345678_24:=FALSE;
ConvStopDly04_24(in:=FALSE);
bQASealingConveyor8:=FALSE;
bQASealingConveyorSample12345678_24:=FALSE;
SealConeMiss:=' Cone  Missing From Sealing Conveyor';
 END_IF
IF bAConeMissAtSealConv8_24 AND bErrorReset THEN
bQASealingConveyor8:=TRUE;  Step4:=5;  tSealStopDly_24:=t#4s;
SealConeMiss:='Continue Machine Operation'; bAConeMissAtSealConv8_24:=FALSE; END_IF

IF bQASealingConveyor8 THEN ConvStopDly04_24(IN:=TRUE , PT:=t#6s , Q=> , ET=> ); bQASealingConveyorSample12345678_24:=TRUE; END_IF
IF ConvStopDly04_24.Q THEN bQASealingConveyor12345678_24:=TRUE; END_IF



									(*##############################Alarm Sequence in HMI#################################*)


IF bAConeMissAtSealConv01_24 OR bAConeMissAtSealConv2_24 OR bAConeMissAtSealConv3_24 OR bAConeMissAtSealConv8_24
OR bAConeMissAtSealConv4_24 OR bAConeMissAtSealConv5_24 OR bAConeMissAtSealConv6_24 OR bAConeMissAtSealConv7_24  THEN
 bQSealBitAlert:=TRUE; END_IF

IF bQSealBitAlert   AND bErrorReset   THEN   bQSealBitAlert:=FALSE; END_IF

IF bQASealingConveyor123_24_1 OR  bQASealingConveyor123_24 OR bQASealingConveyor1234_24_1 OR bQASealingConveyor123456_24_1
OR bQASealingConveyor12345678_24 OR bQASealingConveyorSample12345678_24 OR bQASealingConveyorSample123456_24 OR
 bQASealingConveyorSample1234_24 OR bQASealingConveyorSample123_24 THEN
  bQSealBitAlert_24:=TRUE; ELSE  bQSealBitAlert_24:=FALSE;  END_IF

IF bQASealingConveyor1 OR bQASealingConveyor2 OR bQASealingConveyor3 OR bQASealingConveyor4 OR bQASealingConveyor5 OR
bQASealingConveyor6 OR bQASealingConveyor7 OR bQASealingConveyor8 OR bQASealingConveyor9 OR bQASealingConveyor10 OR
bQASealingConveyor11 OR bQASealingConveyor12   THEN SealConeMissAlet_24:= TRUE; ELSE SealConeMissAlet_24:= FALSE; END_IF



IF NOT bIEmergencySwitch OR bStopHmi  OR bServoOff OR bIMcStop THEN
bQSealBitAlert:=FALSE;
bQSealBitAlert_24:=FALSE;
bACounter_24Reset:=TRUE;
CTU_1.RESET:=TRUE;

bAConeMissAtSealConv01_24:=FALSE;
bAConeMissAtSealConv2_24 :=FALSE;
bAConeMissAtSealConv3_24:=FALSE;
bAConeMissAtSealConv4_24:=FALSE;
bAConeMissAtSealConv5_24:=FALSE;
bAConeMissAtSealConv6_24:=FALSE;
bAConeMissAtSealConv7_24:=FALSE;
bAConeMissAtSealConv8_24:=FALSE;

bQASealingConveyor1:=FALSE;
bQASealingConveyor2:=FALSE;
bQASealingConveyor3:=FALSE;
bQASealingConveyor4:=FALSE;
bQASealingConveyor5:=FALSE;
bQASealingConveyor6:=FALSE;
bQASealingConveyor7:=FALSE;
bQASealingConveyor8:=FALSE;
bQASealingConveyor9:=FALSE;
bQASealingConveyor10:=FALSE;
bQASealingConveyor11:=FALSE;
bQASealingConveyor12:=FALSE;

bQASealingConveyor123_24:=FALSE;
bQASealingConveyor1234_24:=FALSE;
bQASealingConveyor123456_24:=FALSE;
bQASealingConveyor12345678_24:=FALSE;

bQASealingConveyor123_24_1:=FALSE;
 bQASealingConveyor1234_24_1:=FALSE;
 bQASealingConveyor123456_24_1:=FALSE;
 bQASealingConveyor12345678_24_1:=FALSE;

bQASealingConveyorSample123_24 :=FALSE;
bQASealingConveyorSample1234_24 :=FALSE;
bQASealingConveyorSample123456_24 :=FALSE;
bQASealingConveyorSample12345678_24:=FALSE;

bCountLock1_24:=FALSE;
bCountLock2_24:=FALSE;
bCountLock3_24:=FALSE;
bCountLock4_24:=FALSE;
bCountLock5_24:=FALSE;
bCountLock6_24:=FALSE;
bCountLock7_24:=FALSE;
bCountLock8_24:=FALSE;
bCountLock9_24:=FALSE;
bCountLock10_24:=FALSE;
bCountLock11_24:=FALSE;
bCountLock12_24:=FALSE;

bCountLock123_24:=FALSE;
bCountLock1234_24:=FALSE;
bCountLock123456_24:=FALSE;
bCountLock12345678_24:=FALSE;

bCountLock123_24_1:=FALSE;
bCountLock1234_24_1:=FALSE;
bCountLock123456_24_1:=FALSE;
bCountLock12345678_24_1:=FALSE;

bCountLockBit1_24:=FALSE;
bCountLockBit2_24:=FALSE;
bCountLockBit3_24:=FALSE;
bCountLockBit4_24:=FALSE;

Step1:=0;
Step2:=0;
Step3:=0;
Step4:=0;
Step5:=0;

bCountLock_24:=FALSE;

ConvStopDly1(IN:=FALSE);
ConvStopDly2(IN:=FALSE);
ConvStopDly3(IN:=FALSE);
ConvStopDly4(IN:=FALSE);

ConvStopDly01_24(in:=FALSE);
ConvStopDly02_24(in:=FALSE);
ConvStopDly03_24(in:=FALSE);
ConvStopDly04_24(in:=FALSE);
ConvStopDly06_24(in:=FALSE);
ConvStopDly07_24(in:=FALSE);
ConvStopDly08_24(in:=FALSE);
ConvStopDly09_24(in:=FALSE);
ConvStopDly11_24(in:=FALSE);

bSet1Started_24:=FALSE;
bSet2Started_24:=FALSE;
bSet3Started_24:=FALSE;
bSet4Started_24:=FALSE;

bSealConvStart1_24:=FALSE;
bSealConvStart2_24:=FALSE;
bSealConvStart3_24:=FALSE;


bA3ConeCrossed_24:=FALSE;
bA4ConeCrossed_24:=FALSE;
bA6ConeCrossed_24:=FALSE;
bA8ConeCrossed_24:=FALSE;


bA3ConeSealComp:=FALSE;
bA4thConeSealComp:=FALSE;
bA6thConeSealComp:=FALSE;
bA8thConeSealComp:=FALSE;

bA3ConeSealStarted:=FALSE;
bA4thConeSealStarted:=FALSE;
bA6thConeSealStarted:=FALSE;
bA8thConeSealStarted:=FALSE;




ELSE
bACounter_24Reset:=FALSE;
CTU_1.RESET:=FALSE;
END_IF
END_PROGRAM

(* POU ERROR_1, ST *)
PROGRAM ERROR_1
VAR
	bfAlarmbit1: BOOL;
	sAlarmBuffer: ARRAY[1..5] OF STRING;
	sAlarmArray: ARRAY[0..50] OF STRING;
	ifAlarmStep: INT;
	k: INT;
	sAlarmValue: STRING;
	bfAlarmGenerated: BOOL;
	sAlarm1: STRING(80);
	bfAlarmbit2: BOOL;
	bfAlarmbit3: BOOL;
	bfAlarmbit4: BOOL;
	bfAlarmbit5: BOOL;
	sAlarm2: STRING(80);
	sAlarm3: STRING(80);
	sAlarm4: STRING(80);
	sAlarm5: STRING(80) ;
	ifAlarmMoveStep: INT;
	bfReset: BOOL;
	ifAlarmStepClear: INT;
	bClearAlarm: BOOL;
	bDoIndex: BOOL;
	R_TRIG1: R_TRIG;
	Berror: BOOL;




	bRetIUniitAHomeNok: BOOL;
	bRetreivalUnitHomNok: BOOL;
	bRetIUniitBHomeNok: BOOL;
END_VAR
(*============Reteival Unit Error Messages================== *)


	IF bAutoModeOn AND bMCStartInAuto AND bIUnitA_StartPB AND NOT bIUnitA_RowStopperHome AND NOT bUnitARowStopperStarted  THEN bRetIUniitAHomeNok:=TRUE; ELSE  bRetIUniitAHomeNok:=FALSE; END_IF

	IF bAutoModeOn AND bMCStartInAuto AND bIUnitB_StartPB AND NOT bIUnitB_RowStopperHome AND NOT bUnitBRowStopperStarted THEN bRetIUniitBHomeNok:=TRUE; ELSE  bRetIUniitBHomeNok:=FALSE; END_IF

	IF bRetIUniitAHomeNok OR bRetIUniitAHomeNok THEN bRetreivalUnitHomNok:=TRUE; ELSE bRetreivalUnitHomNok:=FALSE; END_IF


















(*

IF bfAlarmbit1 THEN sAlarmBuffer[1]:=sAlarm1;bfAlarmbit1:=FALSE; END_IF
IF bfAlarmbit2 THEN sAlarmBuffer[2]:=sAlarm2;bfAlarmbit2:=FALSE; END_IF
IF bfAlarmbit3 THEN sAlarmBuffer[3]:=sAlarm3;bfAlarmbit3:=FALSE; END_IF
IF bfAlarmbit4 THEN sAlarmBuffer[4]:=sAlarm4;bfAlarmbit4:=FALSE; END_IF
IF bfAlarmbit5 THEN sAlarmBuffer[5]:=sAlarm5;bfAlarmbit5:=FALSE; END_IF
*)
CASE ifAlarmMoveStep OF

	0:	IF sAlarmBuffer[1]<>'' THEN ifAlarmMoveStep:=1;
			ELSIF sAlarmBuffer[2]<>'' THEN ifAlarmMoveStep:=3;
			ELSIF sAlarmBuffer[3]<>'' THEN ifAlarmMoveStep:=5;
			ELSIF sAlarmBuffer[4]<>'' THEN ifAlarmMoveStep:=7;
			ELSIF sAlarmBuffer[5]<>'' THEN ifAlarmMoveStep:=9;
		END_IF

	1:	sAlarmValue:=sAlarmBuffer[1];bfAlarmGenerated:=TRUE;ifAlarmMoveStep:=ifAlarmMoveStep+1;

	2:	IF NOT bfAlarmGenerated AND NOT bfAlarmbit1 THEN sAlarm1:=sAlarmBuffer[1]:='';ifAlarmMoveStep:=0; END_IF

	3:	sAlarmValue:=sAlarmBuffer[2];bfAlarmGenerated:=TRUE;ifAlarmMoveStep:=ifAlarmMoveStep+1;

	4:	IF NOT bfAlarmGenerated THEN sAlarm2:=sAlarmBuffer[2]:='';ifAlarmMoveStep:=0; END_IF

	5:	sAlarmValue:=sAlarmBuffer[3];bfAlarmGenerated:=TRUE;ifAlarmMoveStep:=ifAlarmMoveStep+1;

	6:	IF NOT bfAlarmGenerated THEN sAlarm3:=sAlarmBuffer[3]:='';ifAlarmMoveStep:=0; END_IF

	7:	sAlarmValue:=sAlarmBuffer[4];bfAlarmGenerated:=TRUE;ifAlarmMoveStep:=ifAlarmMoveStep+1;

	8:	IF NOT bfAlarmGenerated THEN sAlarm4:=sAlarmBuffer[4]:='';ifAlarmMoveStep:=0; END_IF

	9:	sAlarmValue:=sAlarmBuffer[5];bfAlarmGenerated:=TRUE;ifAlarmMoveStep:=ifAlarmMoveStep+1;

	10:	IF NOT bfAlarmGenerated THEN sAlarm5:=sAlarmBuffer[5]:='';ifAlarmMoveStep:=0; END_IF

END_CASE






IF bfAlarmGenerated THEN
CASE ifAlarmStep OF

	0: 	k:=50;ifAlarmStep:=ifAlarmStep+1;

	1:	sAlarmArray[k]:=sAlarmArray[k-1];ifAlarmStep:=ifAlarmStep+1;

	2: 	IF NOT (k=1) THEN k:=k-1;ifAlarmStep:=1; ELSE ifAlarmStep:=ifAlarmStep+1; END_IF

	3:	sAlarmArray[0]:=sAlarmValue;ifAlarmStep:=ifAlarmStep+1;

	4:	bfAlarmGenerated:=FALSE;ifAlarmStep:=0;

END_CASE
END_IF
(*
 IF bClearAlarm THEN
FOR i:=0 TO 50 DO
	sAlarmArray[i]:='';
END_FOR
END_IF
*)
IF bFeedinfCylFwdRsError THEN sAlarmBuffer[1]:='chect Cone Feeding Piston Fwd Reed Switdh'; ELSE sAlarmBuffer[1]:=''; END_IF
IF bfAlarmbit2 THEN sAlarmBuffer[2]:=sAlarm2;ELSE sAlarmBuffer[2]:=''; END_IF
IF bfAlarmbit3 THEN sAlarmBuffer[3]:=sAlarm3;ELSE sAlarmBuffer[3]:=''; END_IF
IF bfAlarmbit4 THEN sAlarmBuffer[4]:=sAlarm4;ELSE sAlarmBuffer[4]:=''; END_IF
IF bfAlarmbit5 THEN sAlarmBuffer[5]:=sAlarm5;ELSE sAlarmBuffer[5]:=''; END_IF

IF bfAlarmbit1 OR bfAlarmbit2 OR bfAlarmbit3 OR bfAlarmbit4 OR bfAlarmbit5 THEN
Berror:=TRUE;
ELSE
Berror:=FALSE;
END_IF
END_PROGRAM

(* Visualisation AA
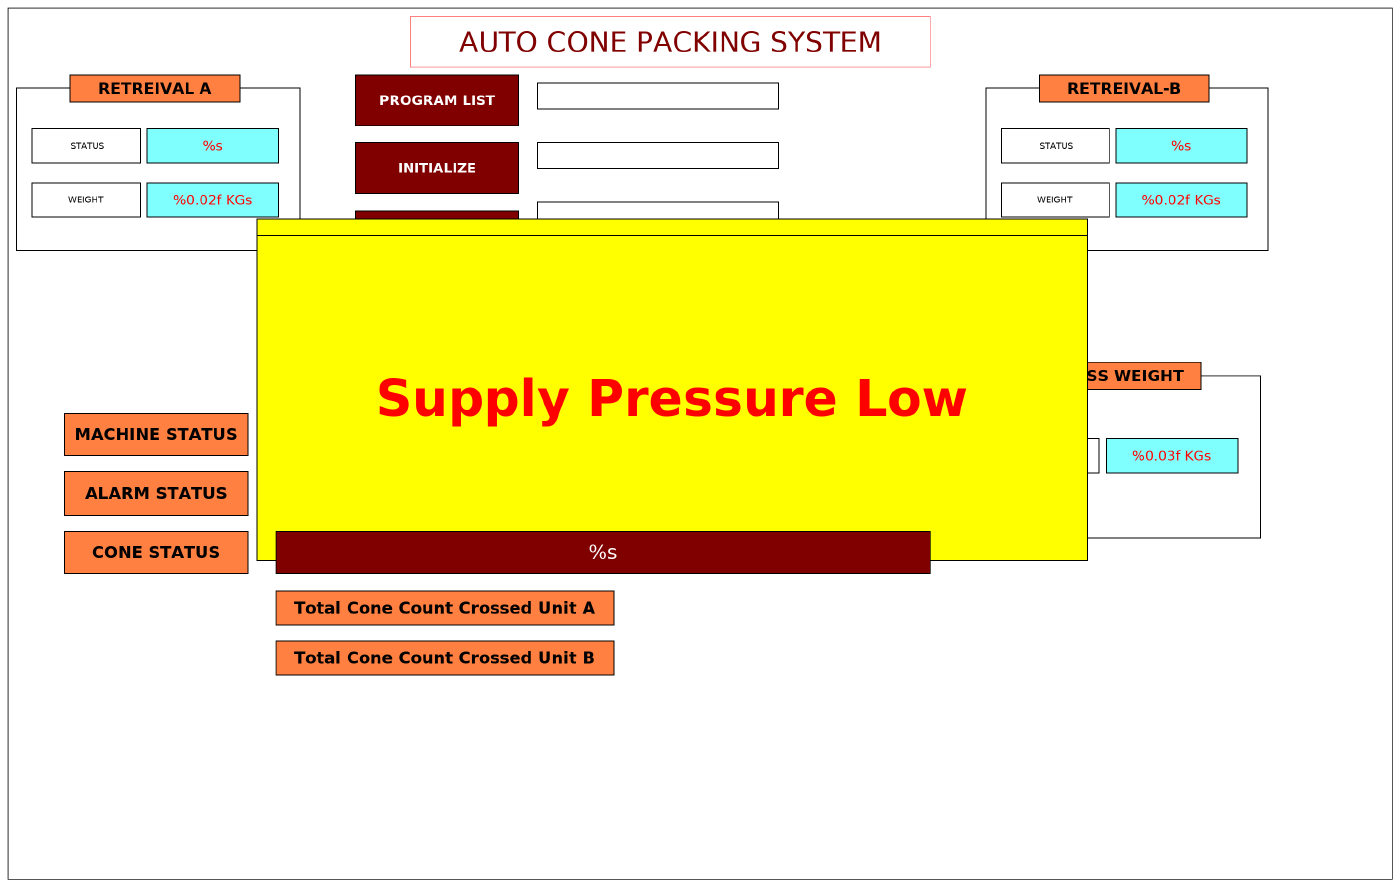
group at (10,0)-(1441,901)
  rounded rectangle at (289,56)-(425,99): text "PROGRAM LIST"; opens Models
  rounded rectangle at (289,113)-(425,156): text "INITIALIZE"; alarm colour if bAInitializeSeq; taps bInitializeHmi
  rounded rectangle at (289,290)-(425,333): text "STOP"; alarm colour if bStopHmi; taps bStopHmi
  rounded rectangle at (440,63)-(641,85): text "PROGRAM NO"
  rounded rectangle at (440,113)-(641,135): text "DETAILS"
  rounded rectangle at (440,163)-(641,185): text "NO OF CONE PROCESSED"
  rounded rectangle at (440,219)-(641,241): text "NO OF CARTONS PROCESSED"
  rounded rectangle at (440,269)-(641,291): text "DATE"
  rounded rectangle at (335,7)-(767,50): text "AUTO CONE PACKING SYSTEM"
  rounded rectangle at (289,170)-(425,213): text "PAUSE"; alarm colour if bAPauseSeq; taps bPauseHmi
  rounded rectangle at (289,226)-(425,270): text "RESUME"; alarm colour if bAPauseSeq; taps bResumeHmi
  rounded rectangle at (47,340)-(200,376): text "MACHINE STATUS"
  rounded rectangle at (47,389)-(200,426): text "ALARM STATUS"
  rounded rectangle at (223,389)-(767,426): text "%s"; shows sMianAlarmStatus
  group at (7,56)-(243,204)
    rounded rectangle at (56,0)-(233,33): text "RETREIVAL A"
    rounded rectangle at (136,64)-(273,105): text "%s"; shows sRetreivalAStatus
    rounded rectangle at (16,64)-(129,105): text "STATUS"
    rounded rectangle at (16,128)-(129,169): text "WEIGHT"
    rounded rectangle at (136,128)-(273,169): text "%0.02f KGs"; shows rRetUnitAWeight
  group at (813,56)-(1048,204)
    rounded rectangle at (56,0)-(233,33): text "RETREIVAL-B"
    rounded rectangle at (136,64)-(273,105): text "%s"; shows sRetreivalBStatus
    rounded rectangle at (16,64)-(129,105): text "STATUS"
    rounded rectangle at (16,128)-(129,169): text "WEIGHT"
    rounded rectangle at (136,128)-(273,169): text "%0.02f KGs"; shows rRetUnitBWeight
  group at (279,248)-(751,397)
    rounded rectangle at (0,0)-(591,211): invisible if not bHidePopUp
    rounded rectangle at (140,110)-(251,161): text "YES"; invisible if NOT bHidePopUp; taps bPauseYesHmi
    rounded rectangle at (320,110)-(431,161): text "NO"; invisible if not bHidePopUp; taps bPauseNoHmi
    rounded rectangle at (88,16)-(513,73): text "Machine is Running. Do You Want to Change / Mode to Manual ?"; invisible if NOT bHidePopUp
    rounded rectangle at (48,168)-(553,201): text "NOTE:- All the Operations will be Aborted."; invisible if NOT bHidePopUp
  rounded rectangle at (223,340)-(767,376): text "%s"; shows sMCStatus
  group at (806,297)-(1042,445)
    rounded rectangle at (56,0)-(233,33): text "GROSS WEIGHT"
    rounded rectangle at (14,91)-(127,132): text "WEIGHT"
    rounded rectangle at (134,91)-(271,132): text "%0.03f KGs"; shows rGrossWeight
  rounded rectangle at (207,177)-(898,450): text "Emergency Pressed"; invisible if NOT bAEmergencyPressed
  rounded rectangle at (207,191)-(898,464): text "Supply Pressure Low"; invisible if NOT bASupplyPressureError
  rounded rectangle at (223,489)-(504,518): text "Total Cone Count Crossed Unit A"
  rounded rectangle at (223,531)-(504,560): text "Total Cone Count Crossed Unit B"
  rounded rectangle at (47,439)-(200,475): text "CONE STATUS"
  rounded rectangle at (223,439)-(767,475): text "%s"; shows Message1_24
4 more shapes without text or variables
*)

(* Visualisation ALARM
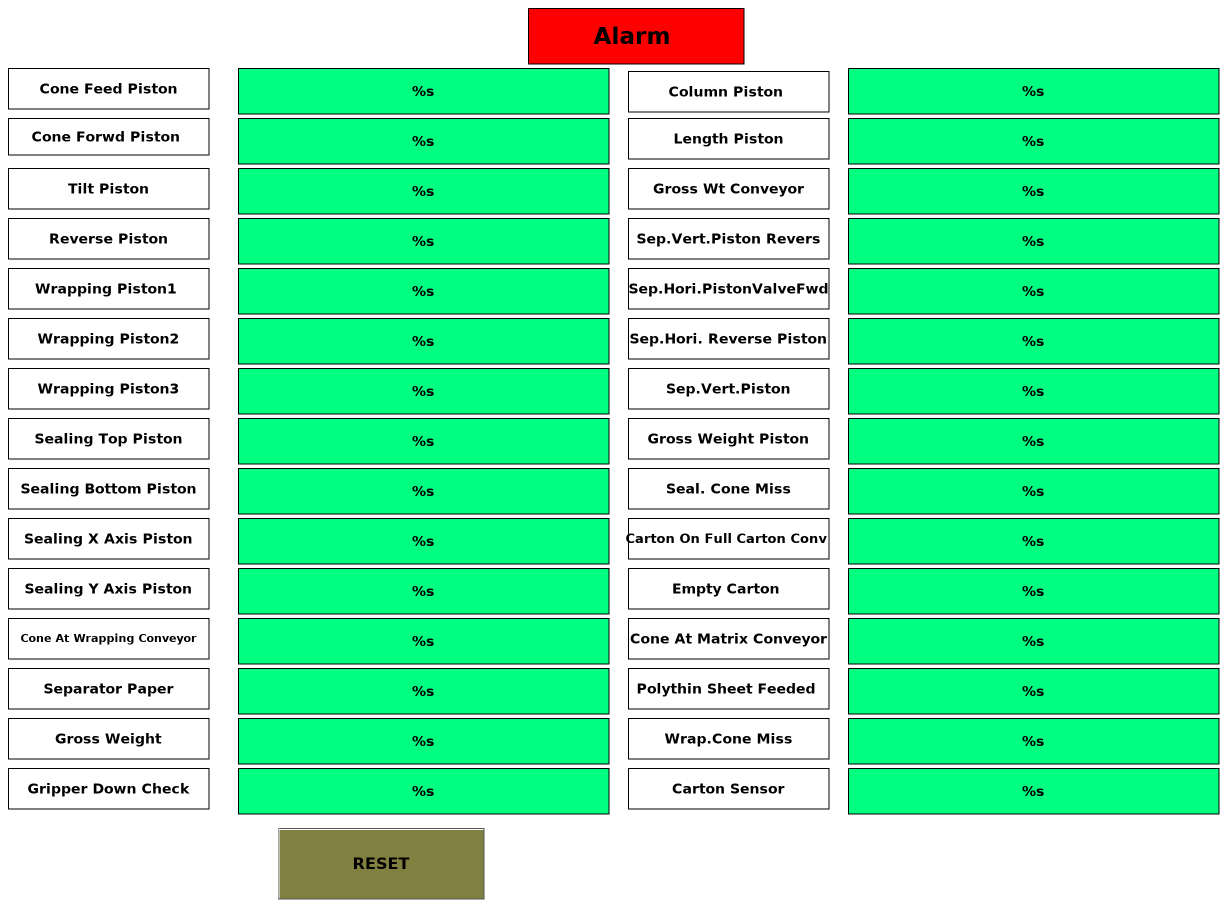
rounded rectangle at (30,100)-(231,137): text "Cone Forwd Piston"
rounded rectangle at (30,50)-(231,91): text "Cone Feed Piston"
rounded rectangle at (30,250)-(231,291): text "Wrapping Piston1"
rounded rectangle at (30,300)-(231,341): text "Wrapping Piston2"
rounded rectangle at (30,350)-(231,391): text "Wrapping Piston3"
rounded rectangle at (30,400)-(231,441): text "Sealing Top Piston"
rounded rectangle at (30,450)-(231,491): text "Sealing Bottom Piston"
rounded rectangle at (30,500)-(231,541): text "Sealing X Axis Piston"
rounded rectangle at (30,550)-(231,591): text "Sealing Y Axis Piston"
rectangle at (260,50)-(631,96): text "%s"; shows .HMIFeedPiston; alarm colour if bAConeFeddCylFwdRsError
rectangle at (260,350)-(631,396): text "%s"; shows .HMIWrapPiston3; alarm colour if bAWrap_3PistRsError
rectangle at (260,300)-(631,346): text "%s"; shows .HMIWrapPiston2; alarm colour if bAWrap_2PistRsError
rectangle at (260,400)-(631,446): text "%s"; shows .HMISealTopPiston; alarm colour if bASealTopPistRsError
rectangle at (260,500)-(631,546): text "%s"; shows .HmiXAxisPiston; alarm colour if bASealSepaX_axisRsError
rectangle at (260,450)-(631,496): text "%s"; shows .HMISealBotPiston; alarm colour if bASealBottomRsError
rectangle at (260,550)-(631,596): text "%s"; shows .HmiYAxisPiston; alarm colour if bASealSepaY_axisRsError
rectangle at (260,250)-(631,296): text "%s"; shows HMIWrapPiston1; alarm colour if bAWrap_1PistRsError
rectangle at (260,100)-(631,146): text "%s"; shows .HMIForwdPiston; alarm colour if bAForwPistRsError
rounded rectangle at (550,-10)-(766,46): text "Alarm"
button at (300,810)-(506,881): text "RESET"; shows .bErrorReset; taps .bErrorReset
rounded rectangle at (30,600)-(231,641): text "Cone At Wrapping Conveyor"
rectangle at (260,600)-(631,646): text "%s"; shows sWrapConvStatus; alarm colour if baConePtrsentAtWrapConv
rounded rectangle at (650,450)-(851,491): text "Seal. Cone Miss"
rectangle at (870,450)-(1241,496): text "%s"; shows .SealConeMiss; alarm colour if SealBitAlert OR bQSealBitAlert
rounded rectangle at (650,500)-(851,541): text "Carton On Full Carton Conv"
rectangle at (870,500)-(1241,546): text "%s"; shows HmiFullCartonAtConveyer; alarm colour if bHmiColourChangeBit
rounded rectangle at (650,53)-(851,94): text "Column Piston"
rounded rectangle at (30,150)-(231,191): text "Tilt Piston"
rounded rectangle at (30,200)-(231,241): text "Reverse Piston"
rounded rectangle at (650,400)-(851,441): text "Gross Weight Piston"
rounded rectangle at (650,300)-(851,341): text "Sep.Hori. Reverse Piston"
rounded rectangle at (650,200)-(851,241): text "Sep.Vert.Piston Revers"
rounded rectangle at (650,350)-(851,391): text "Sep.Vert.Piston"
rounded rectangle at (650,250)-(851,291): text "Sep.Hori.PistonValveFwd"
rectangle at (260,150)-(631,196): text "%s"; shows .HmiTiltPiston; alarm colour if bATiltPistRsError
rectangle at (870,400)-(1241,446): text "%s"; shows .HmiGrossWtPiston; alarm colour if bAGrossWtSenRsError
rectangle at (260,200)-(631,246): text "%s"; shows .HmiReverPiston; alarm colour if bAReversPistnRsError
rectangle at (870,300)-(1241,346): text "%s"; shows .HmiSepHoriRevPiston; alarm colour if bASepaHoriRevValveRsError
rectangle at (870,350)-(1241,396): text "%s"; shows .HmiSepVertiPiston
rectangle at (870,200)-(1241,246): text "%s"; shows .HmiSepVertiPiston; alarm colour if bASepaVertiEndPistnRsError
rectangle at (870,250)-(1241,296): text "%s"; shows .HmiSepHoriRevPiston; alarm colour if bASepaHoriForwdEndRsError
rectangle at (870,50)-(1241,96): text "%s"; shows .HmiColuPushrPiston; alarm colour if bAColumnPushPistnRsError
rounded rectangle at (650,100)-(851,141): text "Length Piston"
rectangle at (870,100)-(1241,146): text "%s"; shows .HmiLengthPiston; alarm colour if bAL_BTightHomeSenRsError
rounded rectangle at (650,150)-(851,191): text "Gross Wt Conveyor"
rectangle at (870,150)-(1241,196): text "%s"; shows sOneMinConMsg; alarm colour if bACartonOnGrossWtConv
rounded rectangle at (650,550)-(851,591): text "Empty Carton"
rectangle at (870,550)-(1241,596): text "%s"; shows HMIEmptyCartonDetectErr; alarm colour if bEmptyCartonDetectError
rounded rectangle at (650,600)-(851,641): text "Cone At Matrix Conveyor"
rectangle at (870,600)-(1241,646): text "%s"; shows sMatrixConvStatus; alarm colour if bAConeMissAtMatricConv
rounded rectangle at (30,650)-(231,691): text "Separator Paper"
rectangle at (260,650)-(631,696): text "%s"; shows HMISeparatorPaperDetec; alarm colour if SeparatorAlertbit
rounded rectangle at (650,650)-(851,691): text "Polythin Sheet Feeded"
rectangle at (870,650)-(1241,696): text "%s"; shows bSheetNotFeeded; alarm colour if bAPolythinSheetError
rounded rectangle at (30,700)-(231,741): text "Gross Weight"
rectangle at (260,700)-(631,746): text "%s"; shows GrossWtAlarm; alarm colour if bGrossWieghtNOk
rounded rectangle at (650,700)-(851,741): text "Wrap.Cone Miss"
rectangle at (870,700)-(1241,746): text "%s"; shows ConeMissAlarm; alarm colour if bHmiColourChangeBit2
rounded rectangle at (650,750)-(851,791): text "Carton Sensor"
rectangle at (870,750)-(1241,796): text "%s"; shows HmiFullCartonAtConveyer_sensor; alarm colour if bHmiColourChangeBit2_24
rounded rectangle at (30,750)-(231,791): text "Gripper Down Check"
rectangle at (260,750)-(631,796): text "%s"; shows sMessage_ServoGripperDown; alarm colour if bAGripperConeAllignError
1 elements of other kinds (tables, trends, ...) not read
*)

(* Visualisation AUTO
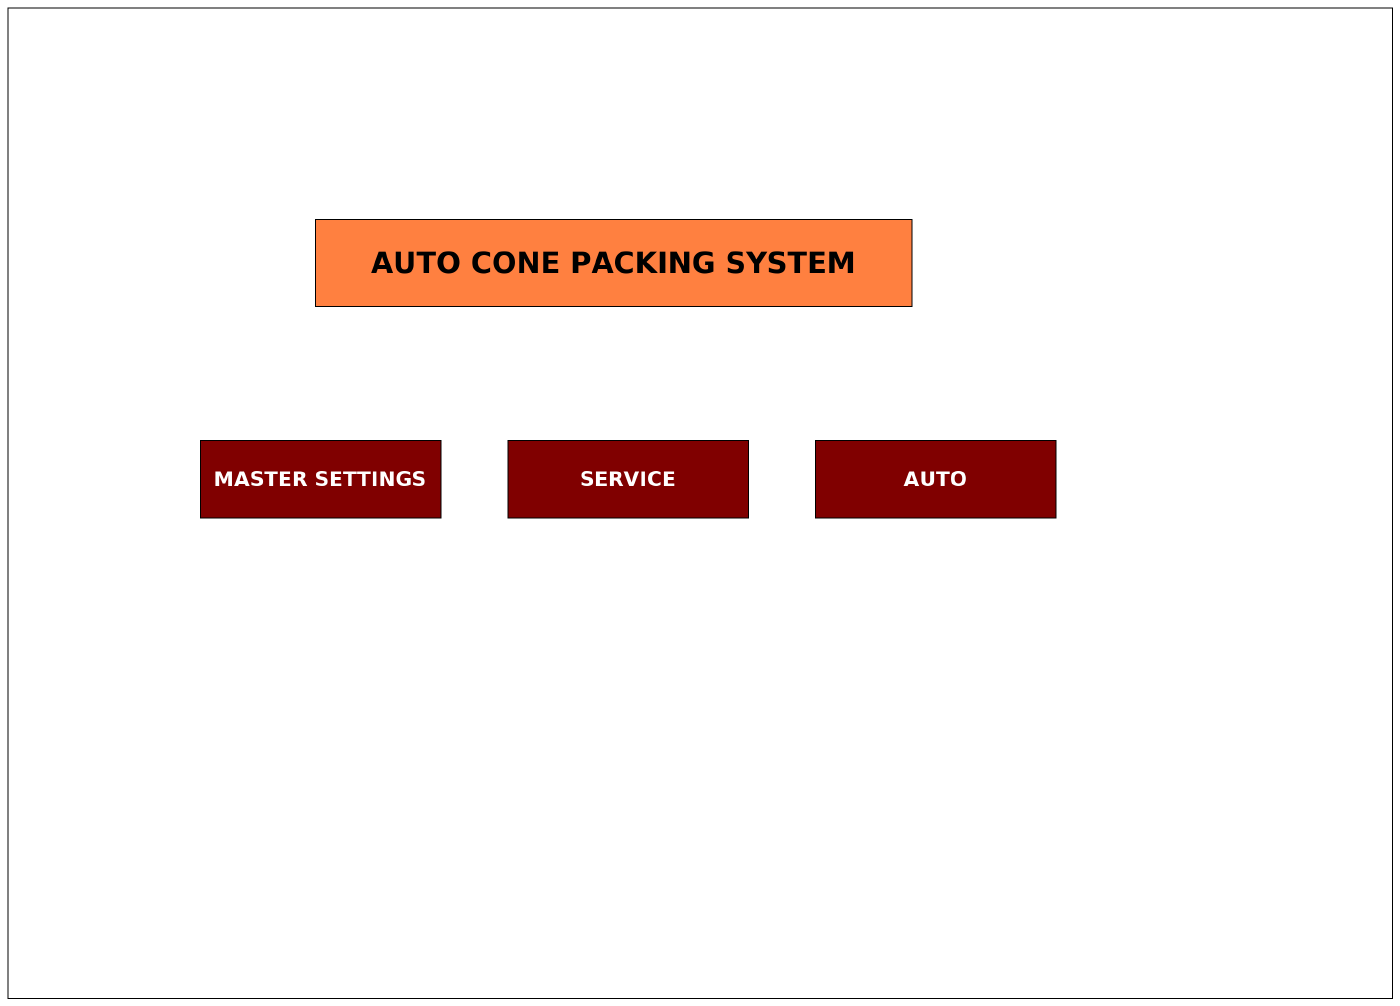
rounded rectangle at (200,450)-(451,531): text "MASTER SETTINGS"; opens MASTER_SETTINGS
rounded rectangle at (520,450)-(771,531): text "SERVICE"; opens SERVICE
rounded rectangle at (840,450)-(1091,531): text "AUTO"; opens AA
rounded rectangle at (320,220)-(941,311): text "AUTO CONE PACKING SYSTEM"
1 more shapes without text or variables
2 elements of other kinds (tables, trends, ...) not read
*)

(* Visualisation BB
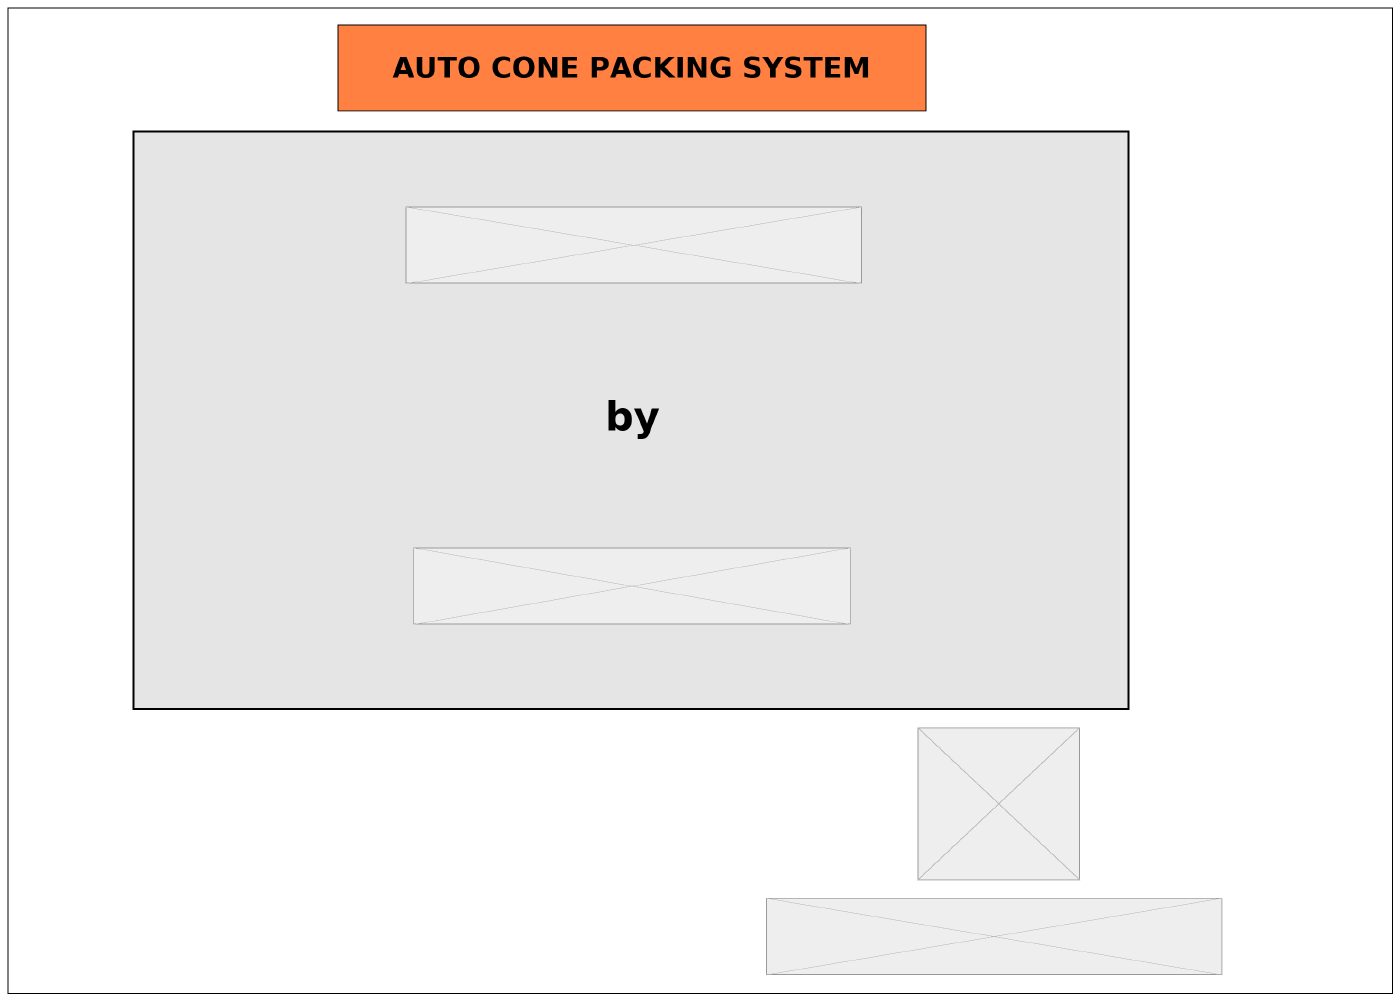
bitmap at (780,930)-(1261,1011): c:\twincat\plc\visu\autocone-logom1.jpg
rounded rectangle at (328,8)-(949,99): text "AUTO CONE PACKING SYSTEM"; invisible if NOT MAIN.EverRunTimer.Q
bitmap at (940,750)-(1111,911): c:\twincat\plc\visu\startbutton.jpg
group at (112,120)-(1169,735)
  rounded rectangle at (0,0)-(1051,611): invisible if MAIN.EverRunTimer.Q
  bitmap at (288,80)-(769,161): c:\twincat\plc\visu\autocone-logom1.jpg
  bitmap at (296,440)-(757,521): c:\twincat\plc\visu\indo_logo1.bmp
  rectangle at (272,256)-(783,347): text "by"
2 more shapes without text or variables
*)

(* Visualisation CONFIGURATION
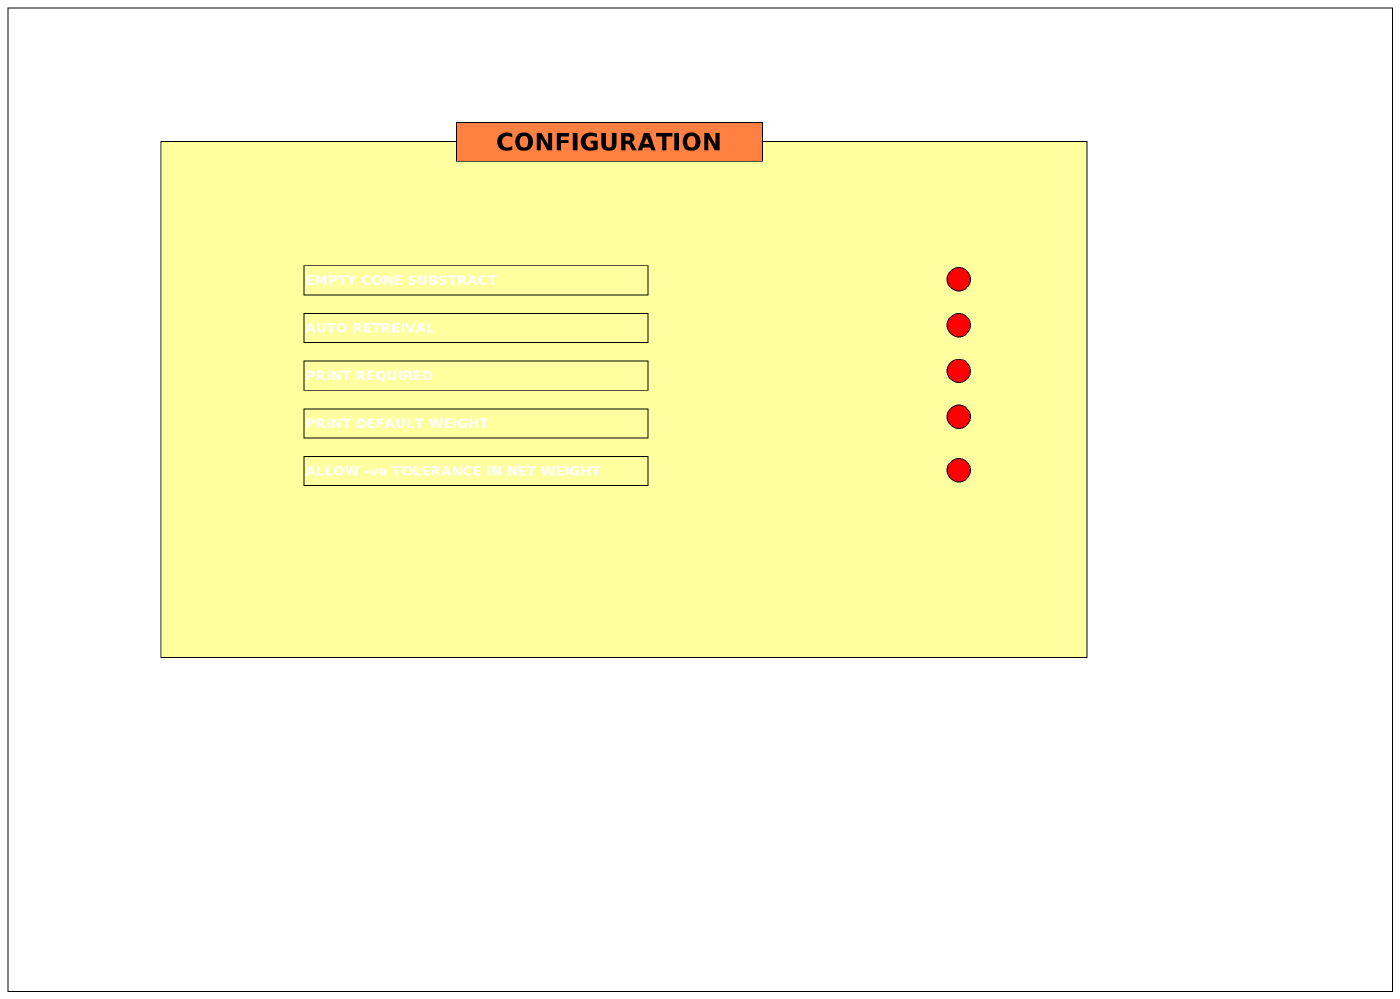
rounded rectangle at (310,270)-(671,301): text "EMPTY CONE SUBSTRACT"
rounded rectangle at (310,320)-(671,351): text "AUTO RETREIVAL"
rounded rectangle at (310,370)-(671,401): text "PRINT REQUIRED"
rounded rectangle at (310,420)-(671,451): text "PRINT DEFAULT WEIGHT"
rounded rectangle at (310,470)-(671,501): text "ALLOW -ve TOLERANCE IN NET WEIGHT"
rounded rectangle at (470,120)-(791,161): text "CONFIGURATION"
ellipse at (984,320)-(1009,345): alarm colour if bAutoRetrivalEnabled
ellipse at (984,272)-(1009,297): alarm colour if bEmptyConeSubEnabled
ellipse at (984,368)-(1009,393): alarm colour if bPrintAutoEnabled
ellipse at (984,416)-(1009,441): alarm colour if PrintDefaultWeightOnEnabled
ellipse at (984,472)-(1009,497): alarm colour if NegToleranceEnabled
2 more shapes without text or variables
14 elements of other kinds (tables, trends, ...) not read
*)

(* Visualisation DIAGNOSTICS
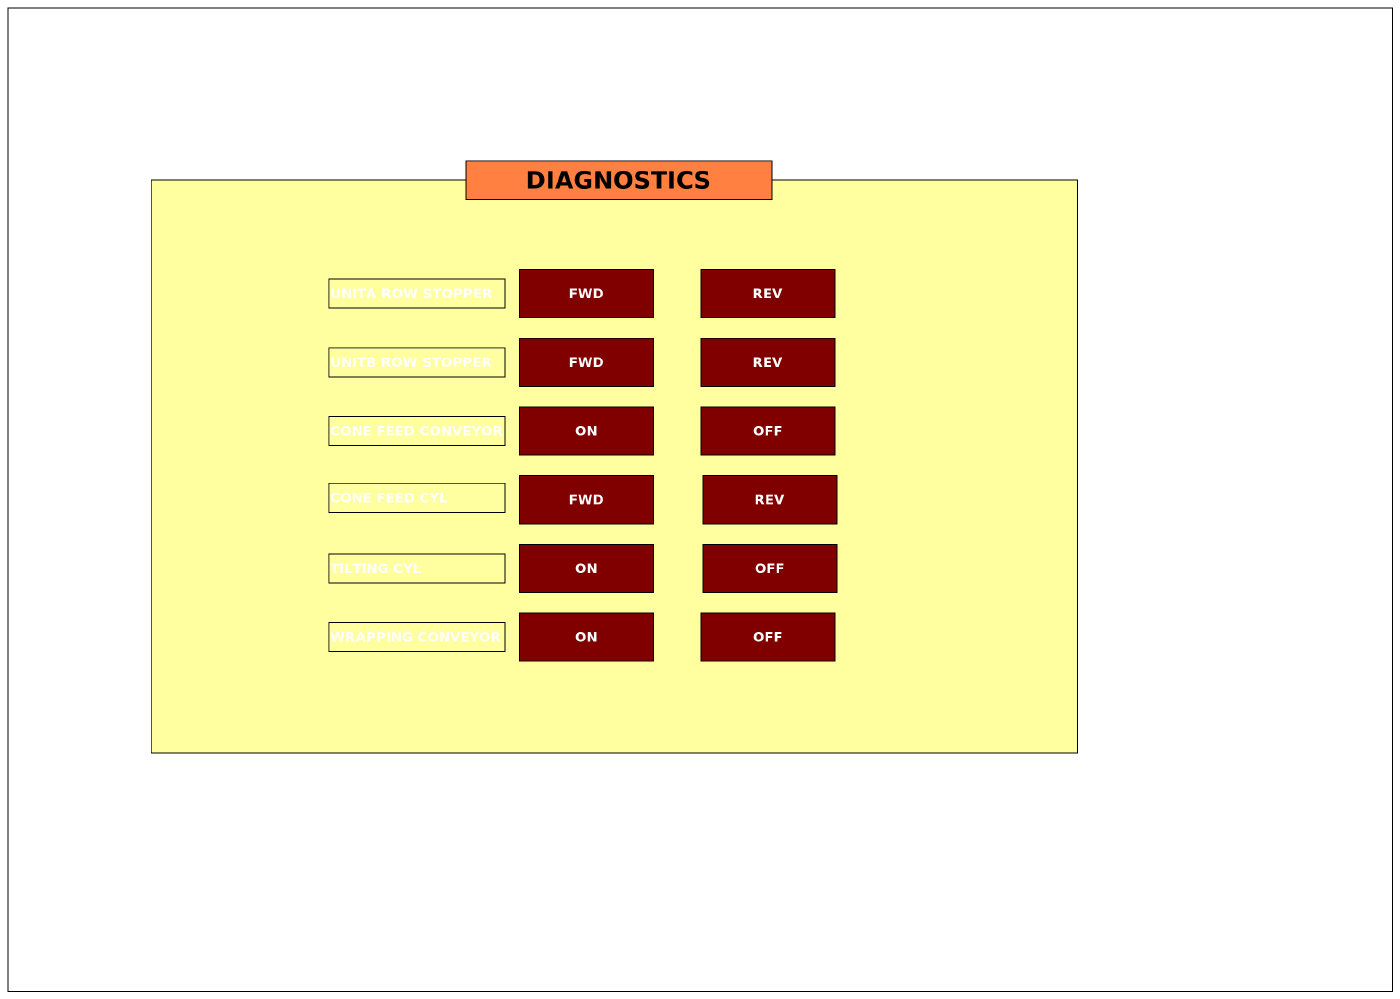
rounded rectangle at (480,70)-(801,111): text "DIAGNOSTICS"
rounded rectangle at (536,184)-(677,235): text "FWD"; alarm colour if .bUA_RowStopperMotorFwdOnHmi; taps .bUA_RowStopperMotorFwdOnHmi
rounded rectangle at (726,184)-(867,235): text "REV"; alarm colour if .bUA_RowStopperMotorRevOnHmi; taps .bUA_RowStopperMotorRevOnHmi
rounded rectangle at (536,256)-(677,307): text "FWD"; alarm colour if .bUB_RowStopperMotorFwdOnHmi; taps .bUB_RowStopperMotorFwdOnHmi
rounded rectangle at (536,328)-(677,379): text "ON"; alarm colour if bFCMotorOnHmi; taps bFCMotorOnHmi
rounded rectangle at (726,256)-(867,307): text "REV"; alarm colour if .bUB_RowStopperMotorRevOnHmi; taps .bUB_RowStopperMotorRevOnHmi
rounded rectangle at (726,328)-(867,379): text "OFF"; alarm colour if bFCMotorOffHmi; taps bFCMotorOffHmi
rounded rectangle at (336,194)-(521,225): text "UNITA ROW STOPPER"
rounded rectangle at (336,266)-(521,297): text "UNITB ROW STOPPER"
rounded rectangle at (336,338)-(521,369): text "CONE FEED CONVEYOR"
rounded rectangle at (536,472)-(677,523): text "ON"; alarm colour if .bCTPistonValveOnHmi; taps .bCTPistonValveOnHmi
rounded rectangle at (728,472)-(869,523): text "OFF"; alarm colour if .bCTPistonValveOffHmi; taps .bCTPistonValveOffHmi
rounded rectangle at (536,400)-(677,451): text "FWD"; alarm colour if .bCFPistonOnHmi; taps .bCFPistonOnHmi
rounded rectangle at (728,400)-(869,451): text "REV"; alarm colour if .bCFPistonOffHmi; taps .bCFPistonOffHmi
rounded rectangle at (336,482)-(521,513): text "TILTING CYL"
rounded rectangle at (336,408)-(521,439): text "CONE FEED CYL"
rounded rectangle at (536,544)-(677,595): text "ON"; alarm colour if .bWCMotorOnHmi; taps .bWCMotorOnHmi
rounded rectangle at (726,544)-(867,595): text "OFF"; alarm colour if .bWCMotorOffHmi; taps .bWCMotorOffHmi
rounded rectangle at (336,554)-(521,585): text "WRAPPING CONVEYOR"
2 more shapes without text or variables
5 elements of other kinds (tables, trends, ...) not read
*)

(* Visualisation DIAGNOSTICS_1
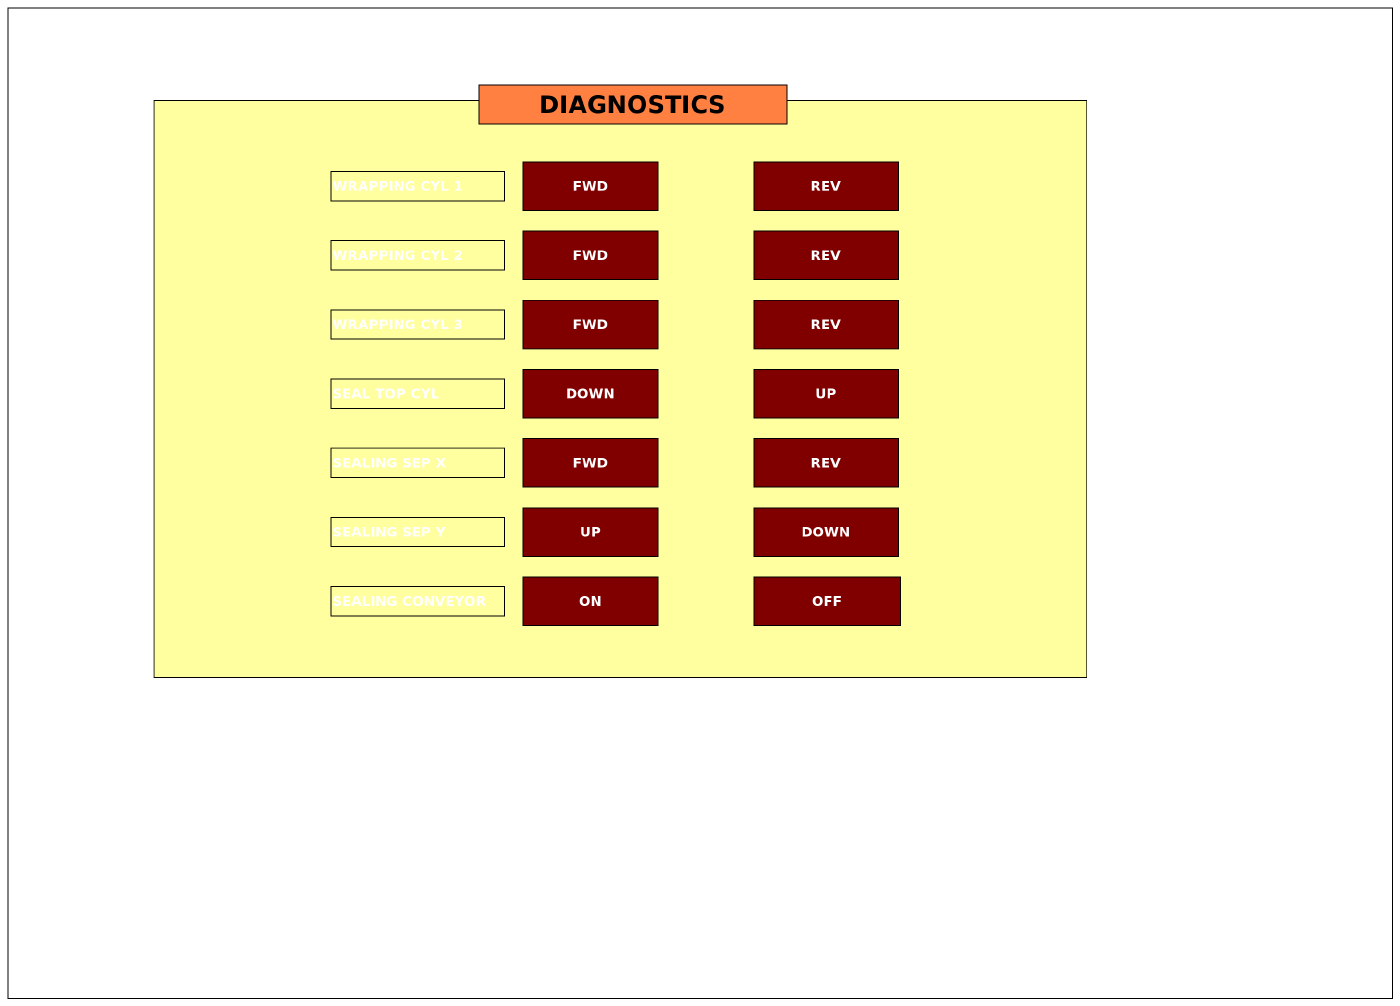
rounded rectangle at (490,80)-(811,121): text "DIAGNOSTICS"
rounded rectangle at (536,160)-(677,211): text "FWD"; alarm colour if .bWrappingCPV1OnHmi; taps .bWrappingCPV1OnHmi
rounded rectangle at (536,232)-(677,283): text "FWD"; alarm colour if .bWrappingCPV2OnHmi; taps .bWrappingCPV2OnHmi
rounded rectangle at (776,232)-(927,283): text "REV"; alarm colour if .bWrappingCPV2OffHmi; taps .bWrappingCPV2OffHmi
rounded rectangle at (536,304)-(677,355): text "FWD"; alarm colour if .bWrappingCPV3OnHmi; taps .bWrappingCPV3OnHmi
rounded rectangle at (776,304)-(927,355): text "REV"; alarm colour if .bWrappingCPV3OffHmi; taps .bWrappingCPV3OffHmi
rounded rectangle at (536,376)-(677,427): text "DOWN"; alarm colour if .bSealingTopPVOnHmi; taps .bSealingTopPVOnHmi
rounded rectangle at (776,376)-(927,427): text "UP"; alarm colour if bSealingTopPVOffHmi; taps bSealingTopPVOffHmi
rounded rectangle at (536,448)-(677,499): text "FWD"; alarm colour if bSSXAxisPistonValveOnHmi; taps bSSXAxisPistonValveOnHmi
rounded rectangle at (776,448)-(927,499): text "REV"; alarm colour if bSSXAxisPistonValveOffHmi; taps bSSXAxisPistonValveOffHmi
rounded rectangle at (336,170)-(517,201): text "WRAPPING CYL 1"
rounded rectangle at (336,242)-(517,273): text "WRAPPING CYL 2"
rounded rectangle at (336,314)-(517,345): text "WRAPPING CYL 3"
rounded rectangle at (336,386)-(517,417): text "SEAL TOP CYL"
rounded rectangle at (336,458)-(517,489): text "SEALING SEP X"
rounded rectangle at (776,160)-(927,211): text "REV"; alarm colour if .bWrappingCPV1OffHmi; taps .bWrappingCPV1OffHmi
rounded rectangle at (536,592)-(677,643): text "ON"; alarm colour if bSCMotorOnHmi; taps bSCMotorOnHmi
rounded rectangle at (776,592)-(929,643): text "OFF"; alarm colour if bSCMotorOffHmi; taps bSCMotorOffHmi
rounded rectangle at (336,602)-(517,633): text "SEALING CONVEYOR"
rounded rectangle at (536,520)-(677,571): text "UP"; alarm colour if bSSYAxisPistonValveOnHmi; taps bSSYAxisPistonValveOnHmi
rounded rectangle at (776,520)-(927,571): text "DOWN"; alarm colour if bSSYAxisPistonValveOffHmi; taps bSSYAxisPistonValveOffHmi
rounded rectangle at (336,530)-(517,561): text "SEALING SEP Y"
2 more shapes without text or variables
5 elements of other kinds (tables, trends, ...) not read
*)

(* Visualisation DIAGNOSTICS_2
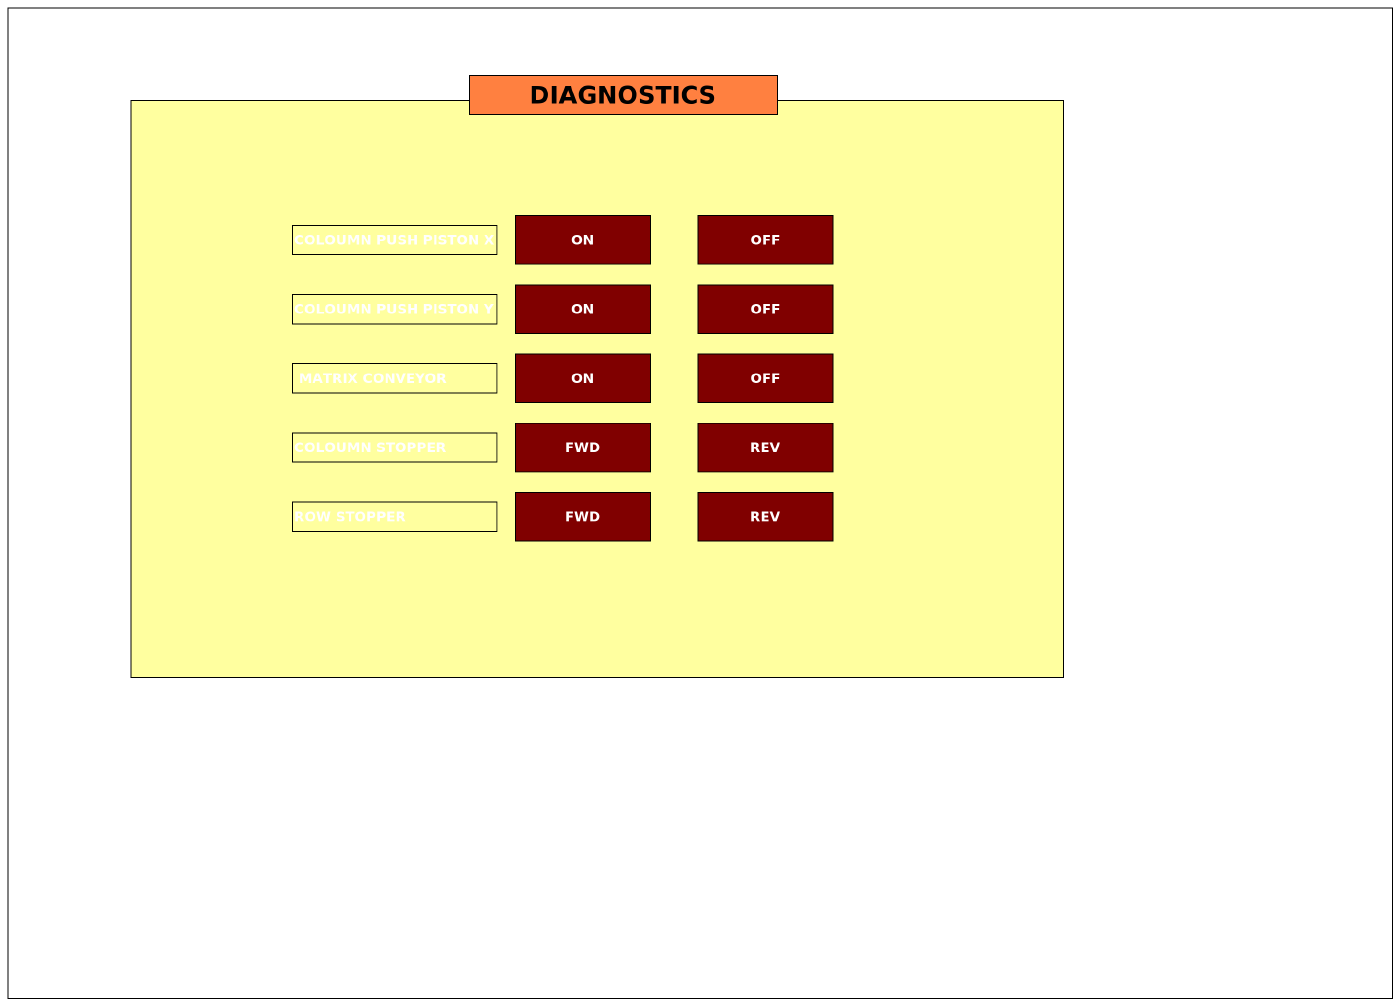
rounded rectangle at (480,70)-(801,111): text "DIAGNOSTICS"
rounded rectangle at (718,360)-(859,411): text "OFF"; alarm colour if .bMCMotorOffHmi; taps .bMCMotorOffHmi
rounded rectangle at (528,360)-(669,411): text "ON"; alarm colour if .bMCMotorOnHmi; taps .bMCMotorOnHmi
rounded rectangle at (296,370)-(509,401): text "MATRIX CONVEYOR"
rounded rectangle at (528,216)-(669,267): text "ON"; alarm colour if bCPushPistonValveOnHmi; taps bCPushPistonValveOnHmi
rounded rectangle at (718,216)-(859,267): text "OFF"; alarm colour if bCPushPistonValveOffHmi; taps bCPushPistonValveOffHmi
rounded rectangle at (296,226)-(509,257): text "COLOUMN PUSH PISTON X"
rounded rectangle at (528,288)-(669,339): text "ON"; alarm colour if bCPushPistonValveYOnHmi; taps bCPushPistonValveYOnHmi
rounded rectangle at (718,288)-(859,339): text "OFF"; alarm colour if bCPushPistonValveYOffHmi; taps bCPushPistonValveYOffHmi
rounded rectangle at (296,298)-(509,329): text "COLOUMN PUSH PISTON Y"
rounded rectangle at (718,432)-(859,483): text "REV"; alarm colour if bCSMotorRevOnHmi; taps bCSMotorRevOnHmi
rounded rectangle at (528,432)-(669,483): text "FWD"; alarm colour if bCSMotorFwdOnHmi; taps bCSMotorFwdOnHmi
rounded rectangle at (296,442)-(509,473): text "COLOUMN STOPPER"
rounded rectangle at (718,504)-(859,555): text "REV"; alarm colour if bRSMotorRevOnHmi; taps bRSMotorRevOnHmi
rounded rectangle at (528,504)-(669,555): text "FWD"; alarm colour if bRSMotorForwardOnHmi; taps bRSMotorForwardOnHmi
rounded rectangle at (296,514)-(509,545): text "ROW STOPPER"
2 more shapes without text or variables
5 elements of other kinds (tables, trends, ...) not read
*)

(* Visualisation DIAGNOSTICS_3
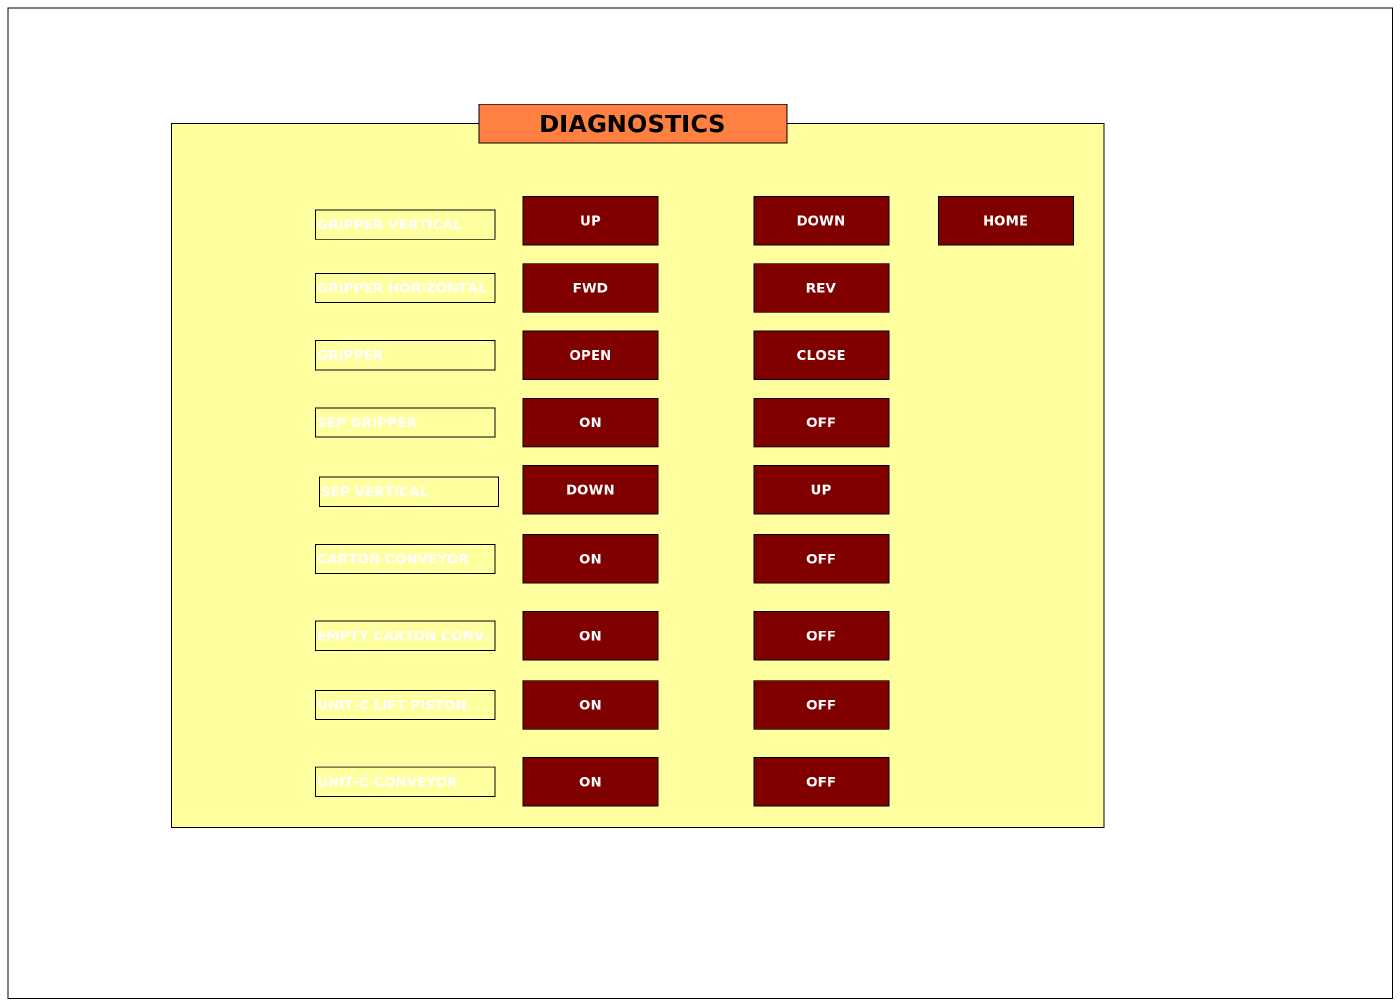
rounded rectangle at (490,80)-(811,121): text "DIAGNOSTICS"
rounded rectangle at (320,190)-(507,221): text "GRIPPER VERTICAL"
rounded rectangle at (320,256)-(507,287): text "GRIPPER HORIZONTAL"
rounded rectangle at (320,326)-(507,357): text "GRIPPER"
rounded rectangle at (320,396)-(507,427): text "SEP GRIPPER"
rounded rectangle at (536,386)-(677,437): text "ON"; alarm colour if bVPValveOnHmi; taps bVPValveOnHmi
rounded rectangle at (776,386)-(917,437): text "OFF"; alarm colour if bVPValveOffHmi; taps bVPValveOffHmi
rounded rectangle at (536,316)-(677,367): text "OPEN"; alarm colour if .bGripperOpenHmi; taps .bGripperOpenHmi
rounded rectangle at (776,316)-(917,367): text "CLOSE"; alarm colour if .bGrippercCloseHmi; taps .bGrippercCloseHmi
rounded rectangle at (536,246)-(677,297): text "FWD"; alarm colour if bSHPistonValveREVOnHmi; taps bSHPistonValveREVOnHmi
rounded rectangle at (776,246)-(917,297): text "REV"; alarm colour if bSHPistonValveOnHmi; taps bSHPistonValveOnHmi
rounded rectangle at (536,176)-(677,227): text "UP"; alarm colour if bJogNegativeHmi; taps bJogNegativeHmi
rounded rectangle at (776,176)-(917,227): text "DOWN"; alarm colour if .bJogPositiveHmi; taps .bJogPositiveHmi
rounded rectangle at (324,468)-(511,499): text "SEP VERTICAL"
rounded rectangle at (536,456)-(677,507): text "DOWN"; alarm colour if bSVPistonValveOnHmi; taps bSVPistonValveOnHmi
rounded rectangle at (776,456)-(917,507): text "UP"; alarm colour if bSVPistonValveOffHmi; taps bSVPistonValveOffHmi
rounded rectangle at (320,538)-(507,569): text "CARTON CONVEYOR"
rounded rectangle at (536,528)-(677,579): text "ON"; alarm colour if bCCMotorOnHmi; taps bCCMotorOnHmi
rounded rectangle at (776,528)-(917,579): text "OFF"; alarm colour if bCCMotorOffHmi; taps bCCMotorOffHmi
rounded rectangle at (320,618)-(507,649): text "EMPTY CARTON CONV."
rounded rectangle at (536,608)-(677,659): text "ON"; alarm colour if bECCMotorOnHmi; taps bECCMotorOnHmi
rounded rectangle at (776,608)-(917,659): text "OFF"; alarm colour if bECCMotorOffHmi; taps bECCMotorOffHmi
rounded rectangle at (320,690)-(507,721): text "UNIT-C LIFT PISTON"
rounded rectangle at (536,680)-(677,731): text "ON"; alarm colour if bGWPistonOnHmi; taps bGWPistonOnHmi
rounded rectangle at (776,680)-(917,731): text "OFF"; alarm colour if bGWPistonOffHmi1; taps bGWPistonOffHmi1
rounded rectangle at (320,770)-(507,801): text "UNIT-C CONVEYOR"
rounded rectangle at (536,760)-(677,811): text "ON"; alarm colour if bRCOnHmi; taps bRCOnHmi
rounded rectangle at (776,760)-(917,811): text "OFF"; alarm colour if bRCOffHmi; taps bRCOffHmi
rounded rectangle at (968,176)-(1109,227): text "HOME"; alarm colour if bServoHomeHmi; taps bServoHomeHmi
2 more shapes without text or variables
4 elements of other kinds (tables, trends, ...) not read
*)

(* Visualisation MASTER_SETTINGS
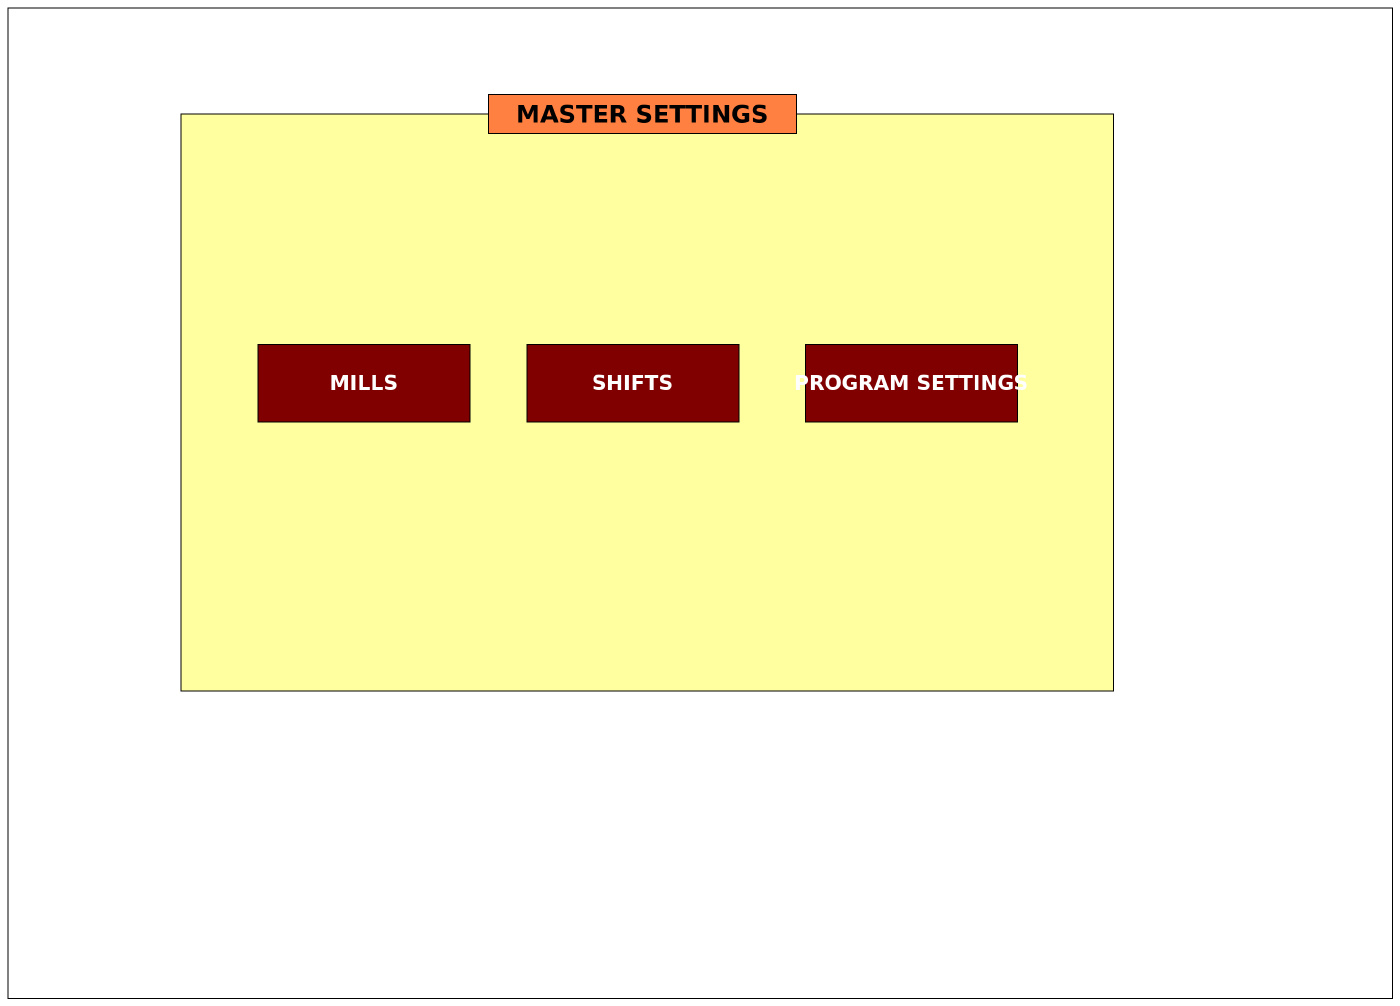
rounded rectangle at (500,90)-(821,131): text "MASTER SETTINGS"
rounded rectangle at (540,350)-(761,431): text "SHIFTS"; opens SHIFT
rounded rectangle at (260,350)-(481,431): text "MILLS"; opens MILL
rounded rectangle at (830,350)-(1051,431): text "PROGRAM SETTINGS"; opens PROGRAM_SETTINGS
2 more shapes without text or variables
4 elements of other kinds (tables, trends, ...) not read
*)

(* Visualisation MILL
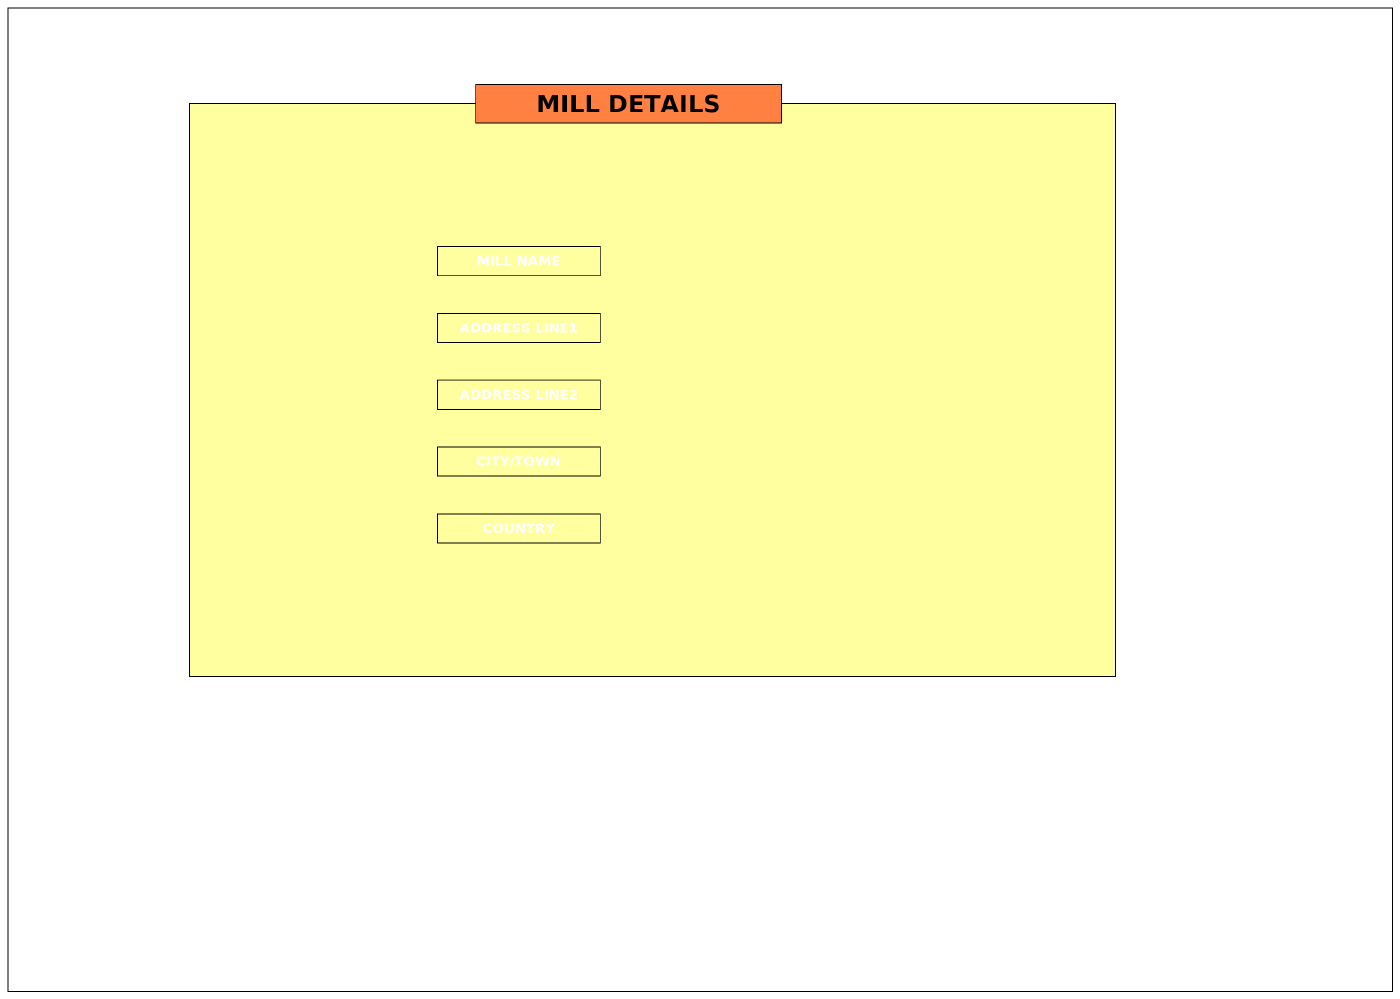
rectangle at (450,250)-(621,281): text "MILL NAME"
rectangle at (450,320)-(621,351): text "ADDRESS LINE1"
rectangle at (450,390)-(621,421): text "ADDRESS LINE2"
rectangle at (450,460)-(621,491): text "CITY/TOWN"
rectangle at (450,530)-(621,561): text "COUNTRY"
rounded rectangle at (490,80)-(811,121): text "MILL DETAILS"
2 more shapes without text or variables
9 elements of other kinds (tables, trends, ...) not read
*)

(* Visualisation MODELS
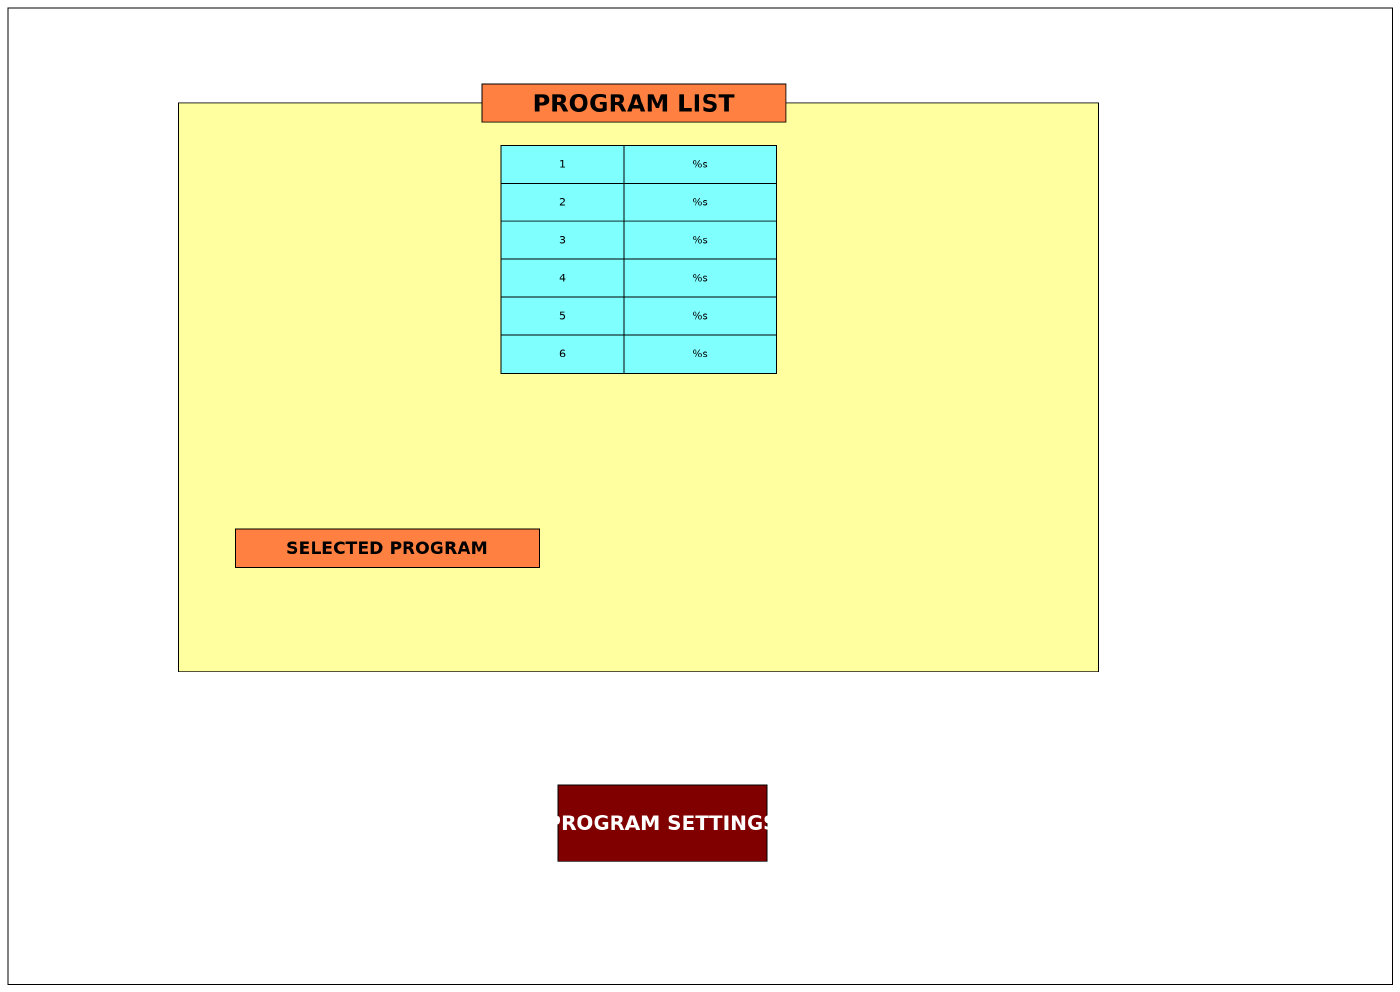
rectangle at (510,145)-(641,186): text "1"; taps bModel1Hmi
rectangle at (640,145)-(801,186): text "%s"; shows PgmNameDis1
rectangle at (510,185)-(641,226): text "2"; taps bModel2Hmi
rectangle at (640,185)-(801,226): text "%s"; shows PgmNameDis2
rectangle at (510,225)-(641,266): text "3"; taps bModel3Hmi
rectangle at (640,225)-(801,266): text "%s"; shows PgmNameDis3
rectangle at (510,265)-(641,306): text "4"; taps bModel4Hmi
rectangle at (640,265)-(801,306): text "%s"; shows PgmNameDis4
rectangle at (510,305)-(641,346): text "5"; taps bModel5Hmi
rectangle at (640,305)-(801,346): text "%s"; shows PgmNameDis5
rectangle at (510,345)-(641,386): text "6"; taps bModel6Hmi
rectangle at (640,345)-(801,386): text "%s"; shows PgmNameDis6
rounded rectangle at (490,80)-(811,121): text "PROGRAM LIST"
rounded rectangle at (230,550)-(551,591): text "SELECTED PROGRAM"
rounded rectangle at (570,820)-(791,901): text "PROGRAM SETTINGS"; opens PROGRAM_SETTINGS
2 more shapes without text or variables
6 elements of other kinds (tables, trends, ...) not read
*)

(* Visualisation PISTON_HOME
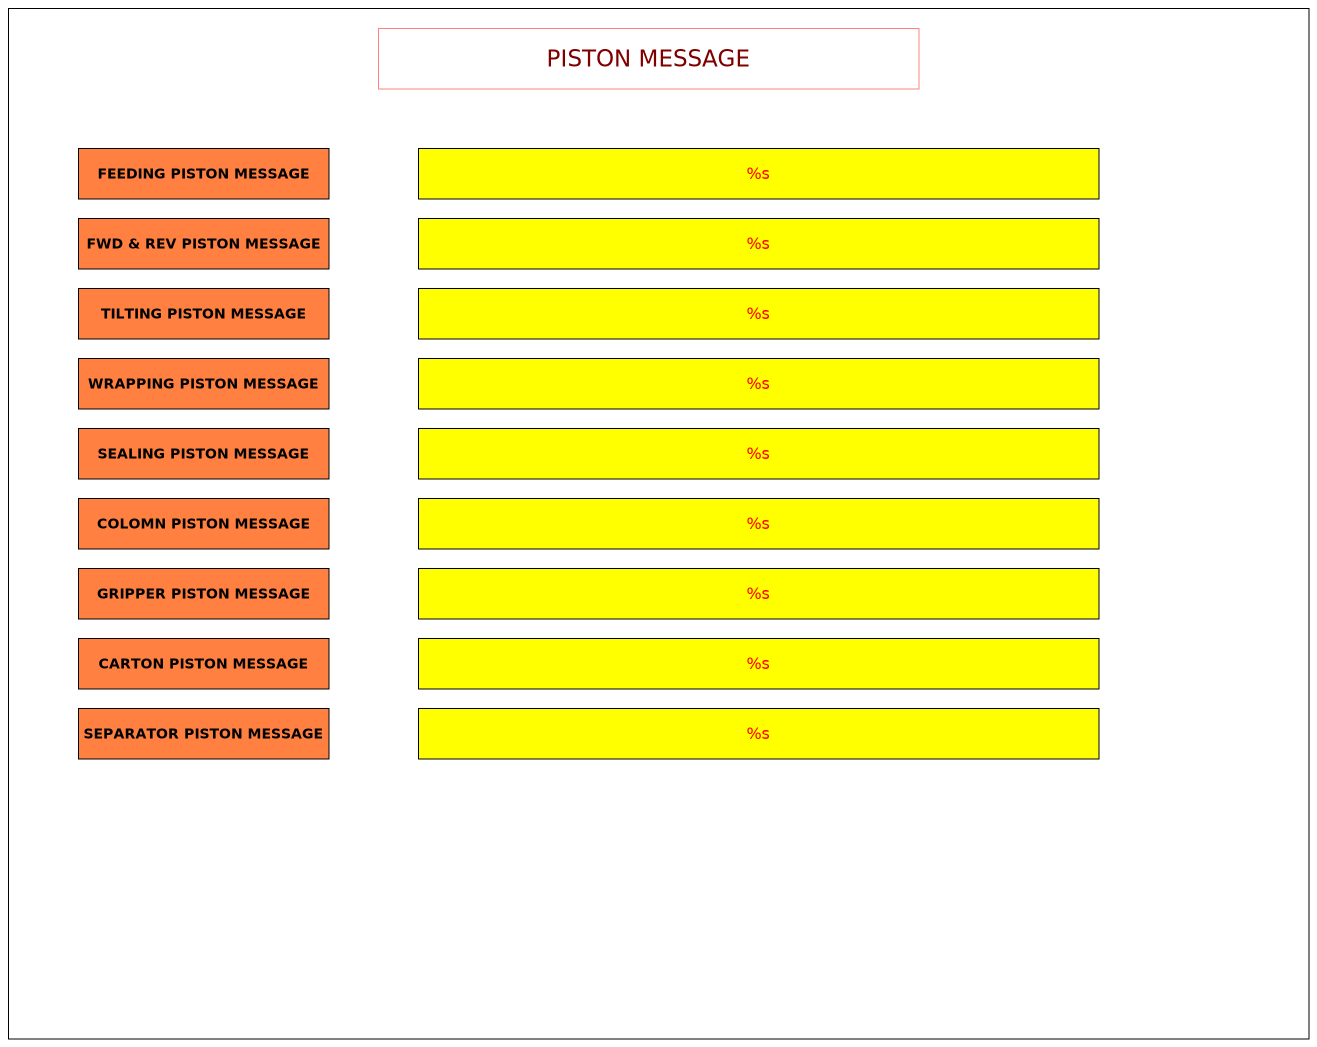
rounded rectangle at (80,150)-(331,201): text "FEEDING PISTON MESSAGE"
rounded rectangle at (80,360)-(331,411): text "WRAPPING PISTON MESSAGE"
rounded rectangle at (80,430)-(331,481): text "SEALING PISTON MESSAGE"
rounded rectangle at (80,500)-(331,551): text "COLOMN PISTON MESSAGE"
rounded rectangle at (80,640)-(331,691): text "CARTON PISTON MESSAGE"
rounded rectangle at (80,570)-(331,621): text "GRIPPER PISTON MESSAGE"
rounded rectangle at (80,710)-(331,761): text "SEPARATOR PISTON MESSAGE"
rounded rectangle at (420,150)-(1101,201): text "%s"; shows sMessage_23_Feeding
rounded rectangle at (420,360)-(1101,411): text "%s"; shows sMessage_Wrapping
rounded rectangle at (420,430)-(1101,481): text "%s"; shows sMessage_Sealing
rounded rectangle at (420,500)-(1101,551): text "%s"; shows sMessage_Colomn
rounded rectangle at (420,570)-(1101,621): text "%s"; shows sMessage_Gripper
rounded rectangle at (420,640)-(1101,691): text "%s"; shows sMessage_Carton
rounded rectangle at (420,710)-(1101,761): text "%s"; shows sMessage_Separator
rounded rectangle at (80,220)-(331,271): text "FWD & REV PISTON MESSAGE"
rounded rectangle at (420,220)-(1101,271): text "%s"; shows sMessage_23_Forwad_rev
rounded rectangle at (420,290)-(1101,341): text "%s"; shows sMessage_23_Tilting
rounded rectangle at (80,290)-(331,341): text "TILTING PISTON MESSAGE"
rounded rectangle at (380,30)-(921,91): text "PISTON MESSAGE"
1 more shapes without text or variables
1 elements of other kinds (tables, trends, ...) not read
*)

(* Visualisation PROGRAM_SETTINGS
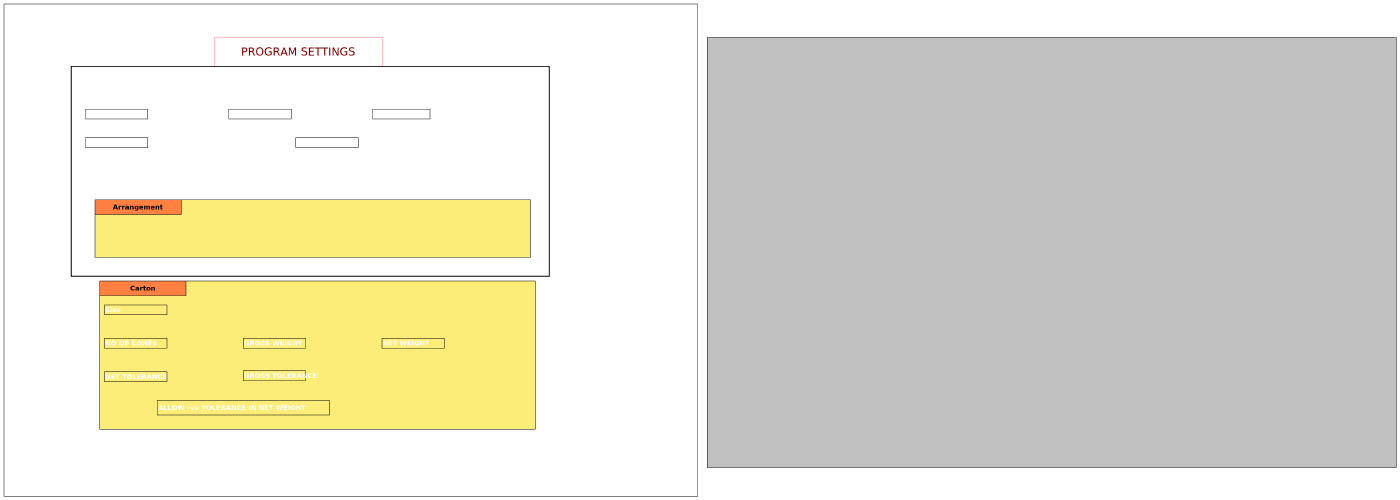
rounded rectangle at (440,0)-(791,61): text "PROGRAM SETTINGS"
rectangle at (200,510)-(381,541): text "Carton"
rounded rectangle at (210,560)-(341,581): text "Size"
rounded rectangle at (210,630)-(341,651): text "NO OF CONES"
rounded rectangle at (500,630)-(631,651): text "GROSS WEIGHT"
rounded rectangle at (790,630)-(921,651): text "NET WEIGHT"
rounded rectangle at (210,700)-(341,721): text "NET TOLERANCE"
rounded rectangle at (500,698)-(631,719): text "GROSS TOLERANCE"
rounded rectangle at (170,150)-(301,171): text "PROGRAM NO"
rounded rectangle at (770,150)-(891,171): text "DETAILS"
rounded rectangle at (470,150)-(601,171): text "COUNT"
rounded rectangle at (170,210)-(301,231): text "LOT NO"
rounded rectangle at (610,210)-(741,231): text "CARTON NO"
rectangle at (190,340)-(371,371): text "Arrangement"
rounded rectangle at (320,760)-(681,791): text "ALLOW -ve TOLERANCE IN NET WEIGHT"
5 more shapes without text or variables
24 elements of other kinds (tables, trends, ...) not read
*)

(* Visualisation RUNNING_STATUS
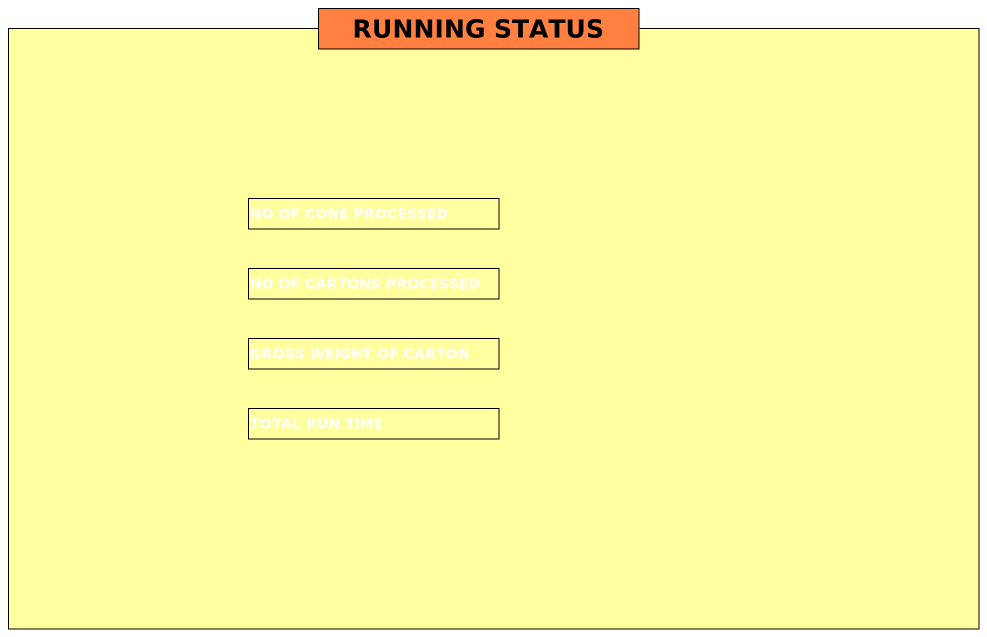
rounded rectangle at (420,280)-(671,311): text "NO OF CONE PROCESSED"
rounded rectangle at (420,350)-(671,381): text "NO OF CARTONS PROCESSED"
rounded rectangle at (420,420)-(671,451): text "GROSS WEIGHT OF CARTON"
rounded rectangle at (420,490)-(671,521): text "TOTAL RUN TIME"
rounded rectangle at (490,90)-(811,131): text "RUNNING STATUS"
1 more shapes without text or variables
7 elements of other kinds (tables, trends, ...) not read
*)

(* Visualisation SERVICE
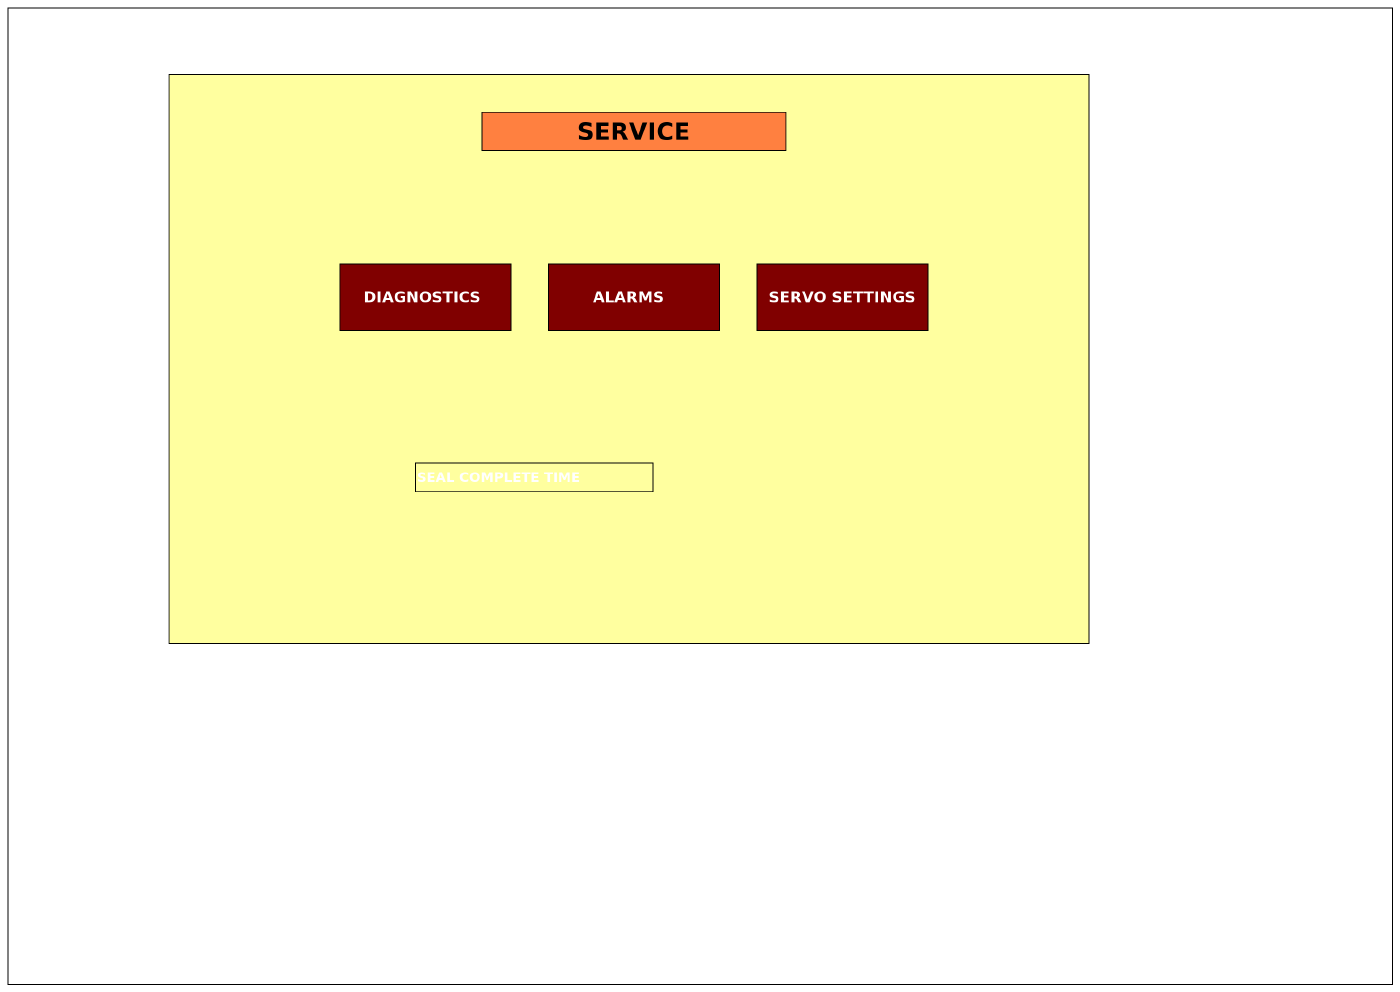
rounded rectangle at (770,270)-(951,341): text "SERVO SETTINGS"; opens Servo
rounded rectangle at (410,480)-(661,511): text "SEAL COMPLETE TIME"
rounded rectangle at (550,270)-(731,341): text "ALARMS"; opens ALARM
rounded rectangle at (330,270)-(511,341): text "DIAGNOSTICS"; opens DIAGNOSTICS
rounded rectangle at (480,110)-(801,151): text "SERVICE"
2 more shapes without text or variables
4 elements of other kinds (tables, trends, ...) not read
*)

(* Visualisation SERVO
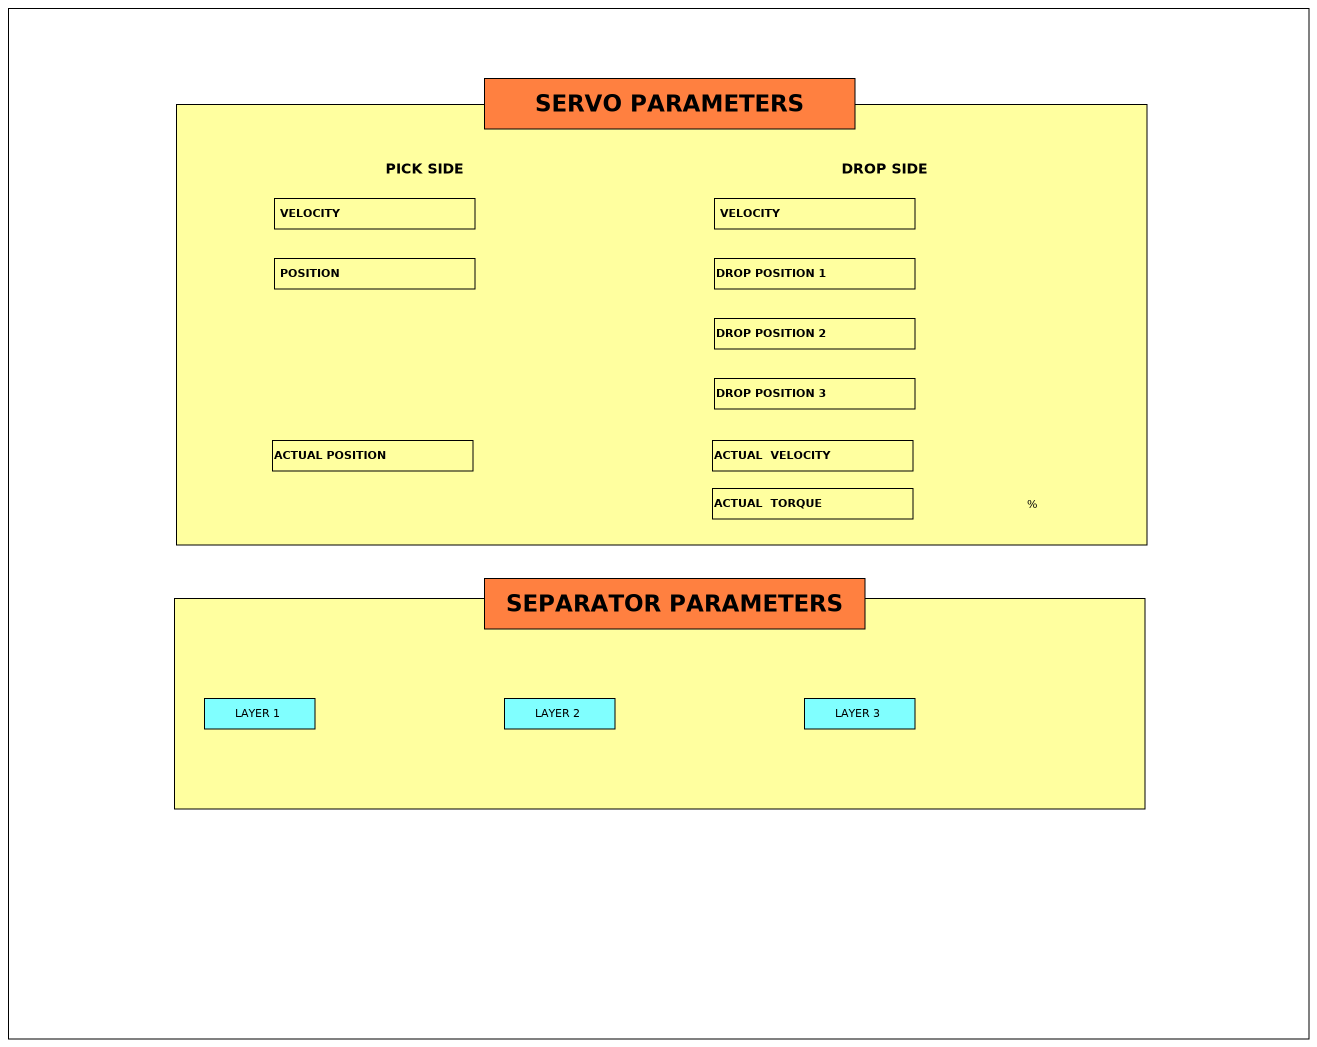
rounded rectangle at (300,140)-(501,181): text "PICK SIDE"
rounded rectangle at (760,140)-(961,181): text "DROP SIDE"
rounded rectangle at (180,690)-(291,721): text "LAYER 1"
rounded rectangle at (480,690)-(591,721): text "LAYER 2"
rounded rectangle at (780,690)-(891,721): text "LAYER 3"
rounded rectangle at (460,70)-(831,121): text "SERVO PARAMETERS"
rounded rectangle at (460,570)-(841,621): text "SEPARATOR PARAMETERS"
rounded rectangle at (250,190)-(451,221): text "VELOCITY"
rounded rectangle at (250,250)-(451,281): text "POSITION"
rounded rectangle at (690,190)-(891,221): text "VELOCITY"
rounded rectangle at (690,250)-(891,281): text "DROP POSITION 1"
rounded rectangle at (690,310)-(891,341): text "DROP POSITION 2"
rounded rectangle at (690,370)-(891,401): text "DROP POSITION 3"
rounded rectangle at (688,432)-(889,463): text "ACTUAL  VELOCITY"
rounded rectangle at (248,432)-(449,463): text "ACTUAL POSITION"
rounded rectangle at (688,480)-(889,511): text "ACTUAL  TORQUE"
rounded rectangle at (984,480)-(1033,513): text "%"
3 more shapes without text or variables
15 elements of other kinds (tables, trends, ...) not read
*)

(* Visualisation SHIFT
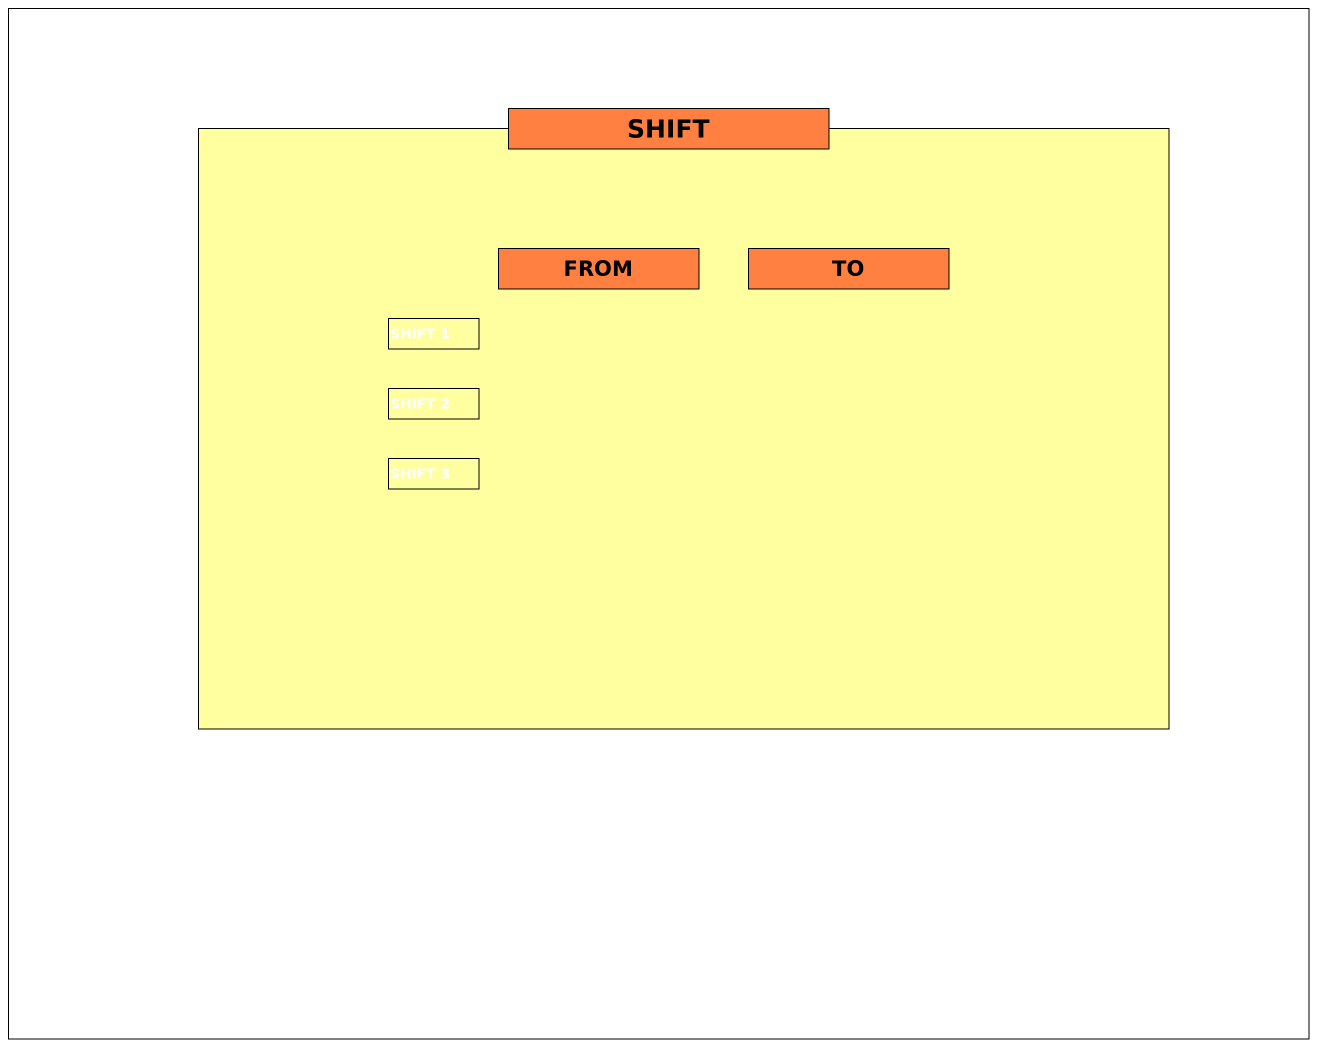
rounded rectangle at (380,310)-(471,341): text "SHIFT 1"
rounded rectangle at (380,380)-(471,411): text "SHIFT 2"
rounded rectangle at (380,450)-(471,481): text "SHIFT 3"
rounded rectangle at (500,100)-(821,141): text "SHIFT"
rounded rectangle at (490,240)-(691,281): text "FROM"
rounded rectangle at (740,240)-(941,281): text "TO"
2 more shapes without text or variables
16 elements of other kinds (tables, trends, ...) not read
*)

(* Visualisation Template
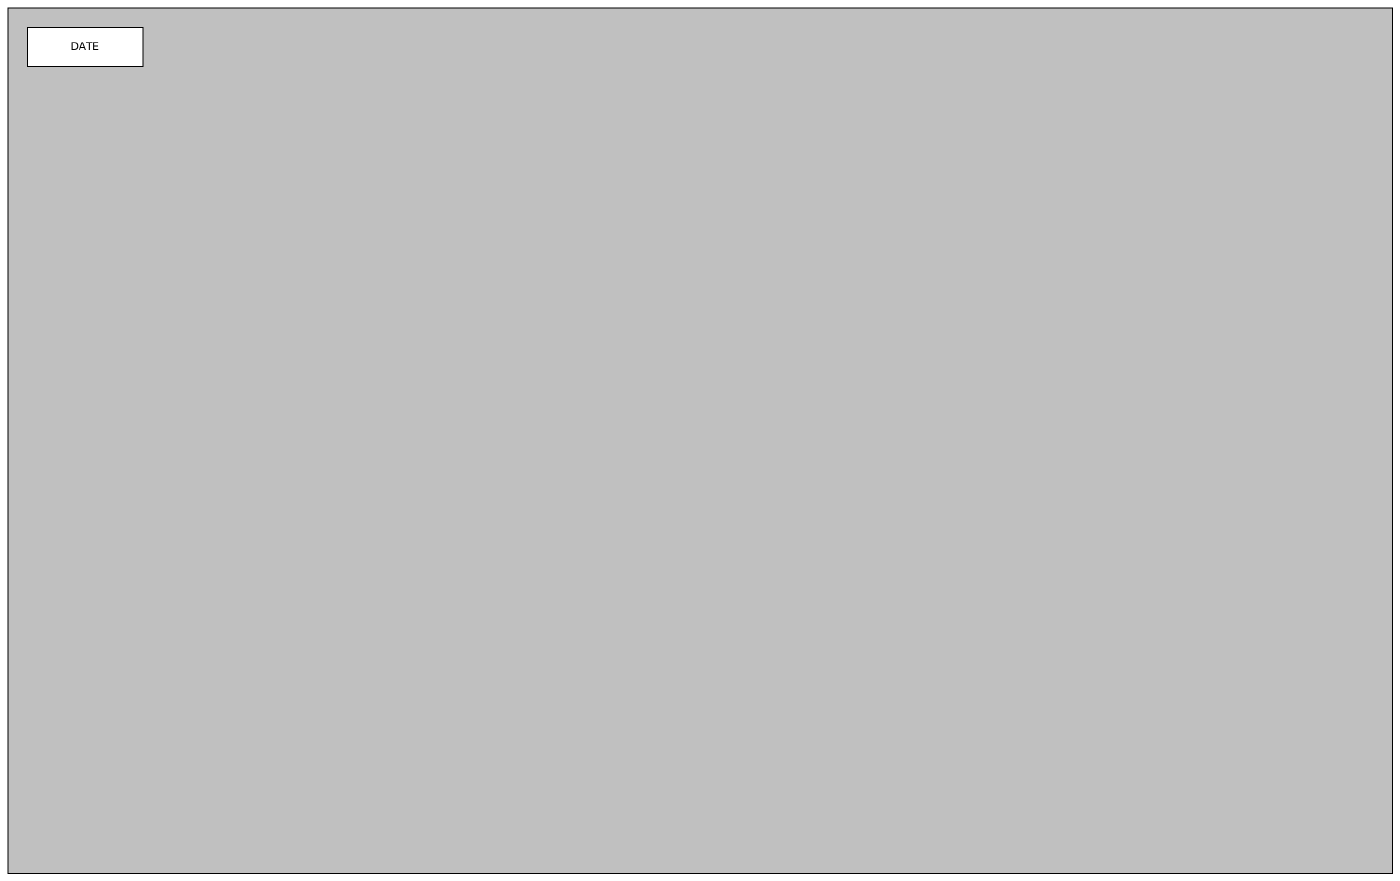
rectangle at (20,20)-(141,61): text "DATE"
1 more shapes without text or variables
*)
